FUNCTION_BLOCK "keller_pressure_transmitters"   // FB99, SCL
{ S7_Optimized_Access := 'TRUE' }
VERSION : 0.1
   VAR_INPUT
      mb_addr : USInt;
   END_VAR
   VAR_IN_OUT
      mb_query : "mb_query";
   END_VAR
   VAR
      sb : "mb_station_block_udt";
      data : Struct
         pressure_sensor_1 : Real;
         pressure_sensor_2 : Real;
         temperature : Real;
         temperature_sensor_1 : Real;
         temperature_sensor_2 : Real;
      END_STRUCT;
   END_VAR
BEGIN
   // Keller, Series 30 and Series 40 - Pressure transmitters
   // 
   // http://www.keller-druck.com/picts/pdf/engl/comm_protocol_e.pdf

   "mb_station_block_header"(sb := #sb,
                             mb_query := #mb_query);

   #mb_query(mb_addr := #mb_addr,
             mode := #mb_query.c.read.holding_reg,
             data_addr := 2,
             data_ptr := #data);

   "mb_station_block_footer"(sb := #sb,
                             mb_query := #mb_query);
END_FUNCTION_BLOCK

FUNCTION_BLOCK "Epever_solar_charge_controller"   // FB109, SCL
{ S7_Optimized_Access := 'TRUE' }
VERSION : 0.1
   VAR_INPUT
      mb_addr : UInt := 1;
      on : Bool;
   END_VAR
   VAR_OUTPUT
      PV_array_input_voltage : Real;
      PV_array_input_current : Real;
      PV_array_input_power : Real;
      battery_power : Real;
      load_voltage : Real;
      load_current : Real;
      load_power : Real;
      battery_temperature : Real;
      temperature_inside_equipment : Real;
      battery_soc : Real;   // The percentage of battery's remaining capacity
      remote_battery_temperature : Real;
      battery_real_rated_power : Real;
      _ : Bool;
      PV_voltage_today_Maximum : Real;
      PV_voltage_today_Minimum : Real;
      Battery_voltage_today_Maximum : Real;
      Battery_voltage_today_Minimum : Real;
      Consumed_energy_today : Real;
      Consumed_energy_this_month : Real;
      Consumed_energy_this_year : Real;
      Consumed_energy_total : Real;
      Generated_energy_today : Real;
      Generated_energy_this_month : Real;
      Generated_energy_this_year : Real;
      Generated_energy_total : Real;
      Battery_voltage : Real;
      Battery_current : Real;
      __ : Bool;
      charging_status : Struct
         No_charging : Bool;
         Float : Bool;
         Boost : Bool;
         Equalization : Bool;
      END_STRUCT;
   END_VAR
   VAR_IN_OUT
      mb_query : "mb_query";
   END_VAR
   VAR
      sb : "mb_station_block_udt";
      read3 : Struct
         load_short : Bool;   // [08]
         load_over_current : Bool;   // [09]
         Input_is_over_current : Bool;   // [10]
         Anti_reverse_MOSFET_is_short : Bool;   // [11]
         Charging_or_Anti_reverse_MOSFET_is_short : Bool;   // [12]
         Charging_MOSFET_is_short : Bool;   // [13]
         x14 : Bool;   // [14]
         x15 : Bool;   // [15]
         Running : Bool;   // [00] - Standby
         Normal : Bool;   // [01] - Fault
         charging_status_0 : Bool;   // [02]
         charging_status_1 : Bool;   // [03]
         PV_Input_is_short : Bool;   // [04]
         x05 : Bool;   // [05]
         x06 : Bool;   // [06]
         Load_MOSFET_is_short : Bool;   // [07]
      END_STRUCT;
      first_scan : Bool := true;
   END_VAR
   VAR_TEMP
      read1 : Struct
         PV_array_input_voltage : UInt;   // [3100]
         PV_array_input_current : UInt;   // [3101]
         PV_array_input_power : UDInt;   // [3102]
         z_1 : Array[1..3] of Word;
         battery_power : UDInt;   // [3106]
         z_2 : Array[1..4] of Word;
         load_voltage : UInt;   // [310C]
         load_current : UInt;   // [310D]
         load_power : UDInt;   // [310E]
         battery_temperature : UInt;   // [3110]
         temperature_inside_equipment : UInt;   // [3111]
         battery_soc : UInt;   // [311A] The percentage of battery's remaining capacity
         remote_battery_temperature : UInt;   // [311B]
         z_3 : UInt;
         battery_real_rated_power : UInt;   // [311D]
      END_STRUCT;
      read2 : Struct
         PV_voltage_today_Maximum : UInt;   // [3300]
         PV_voltage_today_Minimum : UInt;   // [3301]
         Battery_voltage_today_Maximum : UInt;   // [3302]
         Battery_voltage_today_Minimum : UInt;   // [3303]
         Consumed_energy_today : UDInt;   // [3304]
         Consumed_energy_this_month : UDInt;   // [3306]
         Consumed_energy_this_year : UDInt;   // [3308]
         Consumed_energy_total : UDInt;   // [330A]
         Generated_energy_today : UDInt;   // [330C]
         Generated_energy_this_month : UDInt;   // [330E]
         Generated_energy_this_year : UDInt;   // [3310]
         Generated_energy_total : UDInt;   // [3312]
         Battery_voltage : UInt;   // [331A]
         Battery_current : UDInt;   // [331B]
      END_STRUCT;
      tmp : Byte;
   END_VAR
BEGIN
   // Epever - solar charge controller 
   // v2.3 - 12 june 2015
   // 

   IF #first_scan THEN
       #sb.conf.read_only := true;
   END_IF;

   "mb_station_block_header"(sb := #sb, mb_query := #mb_query);
   #mb_query.mb_addr := #mb_addr; 

   #mb_query.mode := #mb_query.c.read.input_reg;
   #mb_query(data_addr := 16#3100, data_ptr := #read1);
   IF #mb_query.Done THEN
       #PV_array_input_voltage := UINT_TO_REAL(#read1.PV_array_input_voltage) / 100;
       #PV_array_input_current := UINT_TO_REAL(#read1.PV_array_input_current) / 100;
       #PV_array_input_power := UDINT_TO_REAL(ROR(IN := #read1.PV_array_input_power, N := 16)) / 100;
       #battery_power := UDINT_TO_REAL(ROR(IN := #read1.battery_power, N := 16)) / 100;
       #load_voltage := UINT_TO_REAL(#read1.load_voltage) / 100;
       #load_current := UINT_TO_REAL(#read1.load_current) / 100;
       #load_power := UDINT_TO_REAL(ROR(IN := #read1.load_power, N := 16)) / 100;
       #battery_temperature := UINT_TO_REAL(#read1.battery_temperature) / 100;
       #temperature_inside_equipment := UINT_TO_REAL(#read1.temperature_inside_equipment) / 100;
       #battery_soc := UINT_TO_REAL(#read1.battery_soc) / 100;
       #remote_battery_temperature := UINT_TO_REAL(#read1.remote_battery_temperature) / 100;
       #battery_real_rated_power := UINT_TO_REAL(#read1.battery_real_rated_power) / 100;
   END_IF;

   #mb_query(data_addr := 16#3300, data_ptr := #read2);
   IF #mb_query.Done THEN
       #PV_voltage_today_Maximum := UINT_TO_REAL(#read2.PV_voltage_today_Maximum) / 100;
       #PV_voltage_today_Minimum := UINT_TO_REAL(#read2.PV_voltage_today_Minimum) / 100;
       #Battery_voltage_today_Maximum := UINT_TO_REAL(#read2.Battery_voltage_today_Maximum) / 100;
       #Battery_voltage_today_Minimum := UINT_TO_REAL(#read2.Battery_voltage_today_Minimum) / 100;
       #Consumed_energy_today := UDINT_TO_REAL(ROR(IN := #read2.Consumed_energy_today, N := 16)) / 100;
       #Consumed_energy_this_month := UDINT_TO_REAL(ROR(IN := #read2.Consumed_energy_this_month, N := 16)) / 100;
       #Consumed_energy_this_year := UDINT_TO_REAL(ROR(IN := #read2.Consumed_energy_this_year, N := 16)) / 100;
       #Consumed_energy_total := UDINT_TO_REAL(ROR(IN := #read2.Consumed_energy_total, N := 16)) / 100;
       #Generated_energy_today := UDINT_TO_REAL(ROR(IN := #read2.Generated_energy_today, N := 16)) / 100;
       #Generated_energy_this_month := UDINT_TO_REAL(ROR(IN := #read2.Generated_energy_this_month, N := 16)) / 100;
       #Generated_energy_this_year := UDINT_TO_REAL(ROR(IN := #read2.Generated_energy_this_year, N := 16)) / 100;
       #Generated_energy_total := UDINT_TO_REAL(ROR(IN := #read2.Generated_energy_total, N := 16)) / 100;
       #Battery_voltage := UDINT_TO_REAL(#read2.Battery_voltage) / 100;
       #Battery_current := UDINT_TO_REAL(ROR(IN := #read2.Battery_current, N := 16)) / 100;
   END_IF;


   #mb_query(data_addr := 16#3201, data_ptr := #read3);
   #tmp.%X0 := #read3.charging_status_0;
   #tmp.%X1 := #read3.charging_status_1;
   #charging_status.No_charging := #tmp = 0;
   #charging_status.Float := #tmp = 1;
   #charging_status.Boost := #tmp = 2;
   #charging_status.Equalization := #tmp = 3;

   #mb_query.mode := #mb_query.c.write.single_discrete_output;
   #tmp.%X0 := #on;
   #mb_query(data_addr := 0, data_ptr := #tmp);

   "mb_station_block_footer"(sb := #sb, mb_query := #mb_query);


   (*
   - 16bit MODBUS addresses (per the modbus.org spec)
   - BPS: 115200 baud
   - Parity: None
   - Data bits: 8
   - Stop bits: 1
   - Flow control: None

   Pin definition RJ45 
   1   Power supply output +7.5
   2   Power supply output +7.5
   3   RS-485 - A
   4   RS-485 - A
   5   RS-485 - B
   6   RS-485 - B
   7   Ground
   8   Ground

   *)
END_FUNCTION_BLOCK

// folder: Library/Modbus/Station blocks/sb untested/Abb

FUNCTION_BLOCK "abb_aquaMaster_3"   // FB4, SCL
{ S7_Optimized_Access := 'TRUE' }
VERSION : 0.1
   VAR_INPUT
      mb_addr : USInt;
   END_VAR
   VAR_IN_OUT
      mb_query : "mb_query";
   END_VAR
   VAR
      sb : "mb_station_block_udt";
      flow : Real;
      pressure : Real;
      totaliser : Struct
         fwd : DInt;
         rev : DInt;
         net : DInt;
      END_STRUCT;
   END_VAR
BEGIN
   // - ABB - AquaMaster 3 - Electromagnetic flowmeter
   // - COI/FET2XX/MOD/TBLÃ¢â‚¬â€œEN
   // - https://library.e.abb.com/public/
   //   91eead459bb0d349c12577fc0033d2b5/COI_FET2XX_MOD_TBL-EN.pdf

   "mb_station_block_header"(sb := #sb, mb_query := #mb_query);
   #mb_query.mb_addr := #mb_addr; // Device address.

   // Two queries, reading input registers. 
   #mb_query.mode := #mb_query.c.read.input_reg;
   #mb_query(data_addr := 5017, data_ptr := #flow);
   #mb_query(data_addr := 5025, data_ptr := #pressure);

   // One query, reading one section of holding registers.
   #mb_query.mode := #mb_query.c.read.holding_reg;
   #mb_query(data_addr := 12003, data_ptr := #totaliser);

   // - Each query reading one section of holding registers.
   // - Data length is automatically calculated for holding 
   //   and input regisers.

   "mb_station_block_footer"(sb := #sb, mb_query := #mb_query);
END_FUNCTION_BLOCK

FUNCTION_BLOCK "Abb_266"   // FB12, SCL
{ S7_Optimized_Access := 'TRUE' }
VERSION : 0.1
   VAR_INPUT
      mb_addr : UInt;
   END_VAR
   VAR_IN_OUT
      mb_query : "mb_query";
   END_VAR
   VAR
      sb : "mb_station_block_udt";
      data : Struct
         "Differential Pressure" : Real;
         "Static Pressure" : Real;
         "Process Temperature" : Real;
         "Mass flow rate value" : Real;
         "Volume Flow rate value" : Real;
      END_STRUCT;
      settings : Struct
         Differential_Pressure_Units_Code : UInt := 12;
         Static_Pressure_Units_select_Code : UInt := 12;
         Temperature_Units_select_Code : UInt := 32;
      END_STRUCT;
   END_VAR
BEGIN
   // ABB - 266 MODBUS, multivariable transmitter.
   // Differential and Static Pressure, Temperature
   // 
   // https://library.e.abb.com/public/9b5a1233ec79400387d5b4887002fb00/2105216MNAA.pdf

   "mb_station_block_header"(sb := #sb, mb_query := #mb_query);
   #mb_query.mb_addr := #mb_addr;

   #mb_query(mode := #mb_query.c.read.holding_reg,
             data_addr := 401,
             data_ptr := #data);

   #mb_query(mode := #mb_query.c.write.holding_reg,
             data_addr := 481,
             data_ptr := #settings);

   "mb_station_block_footer"(sb := #sb, mb_query := #mb_query);

   (*
   Differential_Pressure_Units_Code
   1 = inches of water
   8 = Millibar (ROM default)
   11 = Pascal
   12 = Kilopascal 

   Static Pressure Units select Code
   6 = PSIA
   7 = Bar (ROM default)
   12 = Kilopascal
   117 = Megapascal 

   Temperature Units select Code
   32 = Degree Celsius (ROM default)
   33 = Degree Fahrenheit
   34 = Degree Rankine
   35 = Degree Kelvin

   *)
END_FUNCTION_BLOCK

FUNCTION_BLOCK "Abb_M2M_DMTME"   // FB15, SCL
{ S7_Optimized_Access := 'TRUE' }
VERSION : 0.1
   VAR_INPUT
      mb_addr : UInt;
   END_VAR
   VAR_IN_OUT
      mb_query : "mb_query";
   END_VAR
   VAR
      sb : "mb_station_block_udt";
      read1 : Struct
         "3-PHASE SYSTEM VOLTAGE" : UDInt;   // volt
         voltage_Lx_N : Array[1..3] of UDInt;   // volt
         voltage_L_L : Array[1..3] of UDInt;   // volt 1:L1-L2, 2:L2-L3, 3:L3-L1
         "3-PHASE SYSTEM CURRENT" : UDInt;
         current : Array[1..3] of UDInt;   // mA
         "3-PHASE SYS. POWER FACTOR" : DInt;   // x1000
         Power_factor : Array[1..3] of DInt;   // x1000
         "3-PHASE SYSTEM COS Ï•I" : DInt;   // x1000
         phase_cos : Array[1..3] of DInt;   // x1000
      END_STRUCT;
      read2 : Struct
         "3-PHASE S. APPARENT POWER" : UDInt;   // VA
         apparent_power : Array[1..3] of UDInt;   // VA
         "3-PHASE SYS. ACTIVE POWER" : DInt;   // Watt
         active_power : Array[1..3] of DInt;   // Watt
         "3-PHASE S. REACTIVE POWER" : UDInt;
         reactive_power : Array[1..3] of UDInt;
         "3-PHASE SYS. ACTIVE ENERGY" : UDInt;   // Wh * 100
         "3-PHASE S. REACTIVE ENERGY" : UDInt;   // VArh * 100
         frequency : UDInt;   // mHz
         "MAX LINE CURRENT" : Array[1..3] of UDInt;
      END_STRUCT;
   END_VAR
BEGIN
   // ABB - M2M/DMTME - 2CSG445011D0201 
   //
   // https://library.e.abb.com/public/3921770555944801ad6d9e002d23ca23/2CSG445011D0201.pdf

   "mb_station_block_header"(sb := #sb, mb_query := #mb_query);
   #mb_query.mb_addr := #mb_addr;

   #mb_query.mode := #mb_query.c.read.holding_reg;
   #mb_query(data_addr := 16#1000, data_ptr := #read1);
   #mb_query(data_addr := 16#1026, data_ptr := #read2);

   "mb_station_block_footer"(sb := #sb, mb_query := #mb_query);
END_FUNCTION_BLOCK

FUNCTION_BLOCK "Abb_ach_400_ac_drives"   // FB80, SCL
{ S7_Optimized_Access := 'TRUE' }
VERSION : 0.1
   VAR_INPUT
      mb_addr : UInt;
   END_VAR
   VAR_IN_OUT
      mb_query : "mb_query";
   END_VAR
   VAR
      sb : "mb_station_block_udt";
      read1 : Struct
         sw : Struct   // page 111, tabel 23
            x08_actual_eq_ref : Bool;   // (= is within tolerance limits)
            x09_drive_control_remote : Bool;
            x10_supervision_limit : Bool;   // The value of first supervised parameter equals to or is greater than supervision limit. Refer toGroup 32 Supervision.
            x11_ext2_selected : Bool;   // 0 = ext1 selected
            x12_run : Bool;   // Enable signal received
            x13 : Bool;
            x14 : Bool;
            x15 : Bool;
            x00_rdy_to_sw_on : Bool;
            x01_rdy_to_operate : Bool;
            x02_opr_enabled : Bool;
            x03_falut : Bool;
            x04_OFF2_inactive : Bool;
            x05_OFF3_inactive : Bool;
            x06_switch_on_innhibited : Bool;
            x07_alarm : Bool;   // See the Diagnostics section for a list of relevant alarms
         END_STRUCT;
      END_STRUCT;
      read2 : Struct
         speed : Int;   // rpm
         output_freq : Int;   // 0.1 Hz
         current : Int;   // 0.1 A
         torque : Int;   // 0.1 %
         power : Int;   // 0.1 kW
         dc_bus_voltage : Int;   // 0.1 V
         output_voltage : Int;   // 0.1 V
         ACH400_temp : Int;   // 0.1 Â°C | Displays the temperature of the ACH 400 heatsink in degrees Centigrade
         ext_ref_1 : Int;   // 0.1 Hz
         ext_ref_2 : Int;   // 0.1 %
         ctrl_location : Int;   // 0 - 2
         run_time : UInt;   // h
         kWh_cnt : UInt;   // kWh
         appl_blk_output : UInt;
         digital_input : Struct
            x08 : Bool;
            x09 : Bool;
            x10 : Bool;
            x11 : Bool;
            x12 : Bool;
            x13 : Bool;
            x14 : Bool;
            x15 : Bool;
            x00_in_1 : Bool;
            x01_in_2 : Bool;
            x02_in_3 : Bool;
            x03_in_4 : Bool;
            x04 : Bool;
            x05 : Bool;
            x06 : Bool;
            x07 : Bool;
         END_STRUCT;
         analog_in_1 : UInt;   // 0.1 %
         analog_in_2 : UInt;   // 0.1 %
      END_STRUCT;
      read3 : Struct
         fault_word_1 : Struct
            x08_Motor_overtemperature : Bool;
            x09_Panel_loss : Bool;
            x10_Parameters_inconsistent : Bool;
            x11_DC_bus_ripple_too_large : Bool;
            x12_Motor_stall : Bool;
            x13_Serial_communication_loss : Bool;
            x14_External_fault : Bool;
            x15_Output_ground_fault : Bool;
            x00_Overcurrent : Bool;
            x01_DC_overvoltage : Bool;
            x02_ACH_400_overtemperature : Bool;
            x03_Fault_current : Bool;
            x04_Output_overload : Bool;
            x05_DC_undervoltage : Bool;
            x06_Analog_input_1_fault : Bool;
            x07_Analog_input_2_fault : Bool;
         END_STRUCT;
         fault_word_2 : Struct
            x08_hw_err : Bool;
            x09_hw_err : Bool;
            x10_hw_err : Bool;
            x11_hw_err : Bool;
            x12_hw_err : Bool;
            x13_hw_err : Bool;
            x14_hw_err : Bool;
            x15_hw_err : Bool;
            x00_Underload : Bool;
            x01 : Bool;
            x02_DDCS_link : Bool;
            x03 : Bool;
            x04 : Bool;
            x05 : Bool;
            x06 : Bool;
            x07 : Bool;
         END_STRUCT;
      END_STRUCT;
      _ : Bool;
      write1 : Struct
         cw : Struct   // page 109, tabel 21
            x08 : Bool;
            x09 : Bool;
            x10 : Bool;
            x11_sel_ext_2 : Bool;   // Select external control location 1
            x12 : Bool;
            x13 : Bool;
            x14 : Bool;
            x15 : Bool;
            x00_start : Bool := TRUE;
            x01_no_cost_stop : Bool := TRUE;   // Emergency OFF, coast to stop.Enter OFF2 ACTIVE; proceed to SWITCH-ON INHIBITED
            x02_no_ramp_stop : Bool := TRUE;   // Emergency stop. Drive ramps to stop according to parameter 2205 DECELER TIME 2. Enter
            x03_operation_enable : Bool := TRUE;
            x04 : Bool;
            x05_no_ramp_generator : Bool := TRUE;
            x06_no_force_ramp_generator_input2zero : Bool;   // Force Ramp Function Generator input to zero
            x07_fault_reset : Bool;   // (enter SWITCH-ON INHIBITED)
         END_STRUCT;
         ref_1 : Int;
         ref_2 : Int;
      END_STRUCT;
      write2 : Struct
         keypad_ref_sel : UInt;
         ext1_ext2_sel : UInt;
         ext1_sel : UInt;
         ext1_sel_min : UInt;   // 0 - 250 Hz
         ext1_sel_max : UInt := 50;   // 0 - 250 Hz
      END_STRUCT;
      write3 : Struct   // Communication fault function
         comm_fault_func : UInt := 1;   // 1=FAULT(cost), 2=CONST SP 7, 3=LAST SPEED
      END_STRUCT;
   END_VAR
BEGIN
   // Abb - ACH 400 - AC Drives 
   // 
   // Web: https://www.ccontrols.com/support/dp/ACH402_US_04_Web.pdf

   "mb_station_block_header"(sb := #sb, mb_query := #mb_query);
   #mb_query.mb_addr := #mb_addr;

   #mb_query.mode := #mb_query.c.read.holding_reg;
   #mb_query(data_addr := 3, data_ptr := #read1);   // 40004
   #mb_query(data_addr := 102, data_ptr := #read2); // 103
   #mb_query(data_addr := 304, data_ptr := #read3); // 305 - 1 

   #mb_query.mode := #mb_query.c.write.holding_reg;
   #mb_query(data_addr := 0, data_ptr := #write1); // 40001
   // #mb_query(data_addr := 1100, data_ptr := #write2); // 1101 - 1
   #mb_query(data_addr := 5003, data_ptr := #write3); // 5004 - 1

   "mb_station_block_footer"(sb := #sb, mb_query := #mb_query);
END_FUNCTION_BLOCK

// folder: Library/Modbus/Station blocks/sb untested/Floridan

FUNCTION_BLOCK "Floridan_Uniflo_1200"   // FB83, SCL
{ S7_Optimized_Access := 'TRUE' }
VERSION : 0.1
   VAR_INPUT
      mb_addr : USInt;
      delay : Time := T#10S;
   END_VAR
   VAR_OUTPUT
      energi : LReal;   // [MJ]
      vol_measured : LReal;   // [m3]
      vol_conv : LReal;   // [Nm3]
      pressure : LReal;   // [bar A]
      temperature : LReal;
   END_VAR
   VAR_IN_OUT
      mb_query : "mb_query";
   END_VAR
   VAR
      sb : "mb_station_block_udt";
      battery_remaining : UInt;
      mb_delay : "mb_delay";
      serial_number : String[6];
   END_VAR
   VAR_TEMP
      dommy : Bool;
      c : Int;
      "dword" : DWord;
   END_VAR
BEGIN
   // Flonidan - Uniflo 1200 GVEC
   // Product number: 061864X-YYY
   //
   // - https://www.gavilar.nl/files/communicationboard230210_1521630740_b6a3b533.pdf
   // - M/06180XX/24

   "mb_station_block_header"(sb := #sb, mb_query := #mb_query);
   #mb_query.mb_addr := #mb_addr; // Device address.

   // Reduce power consumption, by halting execution. Nice if the device is running 
   // on battery. mb_delay is located inside the mb_extended_features.scl file.
   #mb_delay(delay := #delay, mb_query := #mb_query);

   #mb_query.mb_addr.%X5 := 0; // - Last bits of mb_addr is used for expanding 
   #mb_query.mb_addr.%X6 := 0; //   register addr, this means that only addr 1
   #mb_query.mb_addr.%X7 := 0; //   to 31 on the bus may be used.

   #mb_query.mode := #mb_query.c.read.holding_reg;

   #mb_query(data_addr := 123, data_ptr := #battery_remaining);
   #mb_query(data_addr := 2833, data_ptr := #serial_number); // Serial number 

   #mb_query.conf.buffer_handler := false;

   #mb_query(data_addr := 56, data_len := 44, data_ptr := #dommy);
   IF #mb_query.Done THEN
       #vol_conv := "intreal"(mb_query := #mb_query, addr := 16#70 / 2);
       #"dword".%B3 := #mb_query.z.buffer[16]; // 16#80/2=64, (64-56)*2=16
       #"dword".%B2 := #mb_query.z.buffer[17];
       #"dword".%B1 := #mb_query.z.buffer[18];
       #"dword".%B0 := #mb_query.z.buffer[19];
       #pressure := DWORD_TO_REAL(#"dword");
       #"dword".%B3 := #mb_query.z.buffer[20]; // 16#84/2=66, (66-56)*2=20
       #"dword".%B2 := #mb_query.z.buffer[21];
       #"dword".%B1 := #mb_query.z.buffer[22];
       #"dword".%B0 := #mb_query.z.buffer[23];
       #temperature := DWORD_TO_REAL(#"dword");
       #energi := "intreal"(mb_query := #mb_query, addr := 16#90 / 2);
       #vol_measured := "intreal"(mb_query := #mb_query, addr := 16#98 / 2);
   END_IF;

   #mb_query.data_len := #mb_query.c.auto_len;
   #mb_query.conf.buffer_handler := true;
   "mb_station_block_footer"(sb := #sb, mb_query := #mb_query);
END_FUNCTION_BLOCK

FUNCTION "intreal" : LReal   // FC16, SCL
{ S7_Optimized_Access := 'TRUE' }
VERSION : 0.1
   VAR_INPUT
      mb_query : "mb_query";
      addr : UInt;
   END_VAR
   VAR_TEMP
      dw : UDInt;
      r : DWord;
      bo : UDInt;
   END_VAR
BEGIN
   // Uniflo 1200 has a special datatype named
   // int-real, this block decode that data type.

   // buffer offset
   #bo := (#addr - #mb_query.data_addr) * 2;

   // The integer part of the value, little endian.
   #dw.%B3 := #mb_query.z.buffer[#bo + 0];
   #dw.%B2 := #mb_query.z.buffer[#bo + 1];
   #dw.%B1 := #mb_query.z.buffer[#bo + 2];
   #dw.%B0 := #mb_query.z.buffer[#bo + 3];
   #intreal := UDINT_TO_LREAL(#dw);

   // The decimal part of the value, little endian.
   // Stored as a real (IEEE754).
   #r.%B3 := #mb_query.z.buffer[#bo + 4];
   #r.%B2 := #mb_query.z.buffer[#bo + 5];
   #r.%B1 := #mb_query.z.buffer[#bo + 6];
   #r.%B0 := #mb_query.z.buffer[#bo + 7];
   #intreal += DWORD_TO_REAL(#r);
END_FUNCTION

// folder: Library/Modbus/Station blocks/sb untested/Grundfoss

FUNCTION_BLOCK "Grunnfoss_pump"   // FB14, SCL
{ S7_Optimized_Access := 'TRUE' }
VERSION : 0.1
   VAR_INPUT
      mb_addr : USInt;
      setpoint : Real;   // [%]
   END_VAR
   VAR_OUTPUT
      ProcessFeedback : Real;
      _ : Bool;
      Head : Real;   // bar
      VolumeFlow : Real;   // m3/h
      RelativePerformance : Real;   // %
      Speed : Real;   // rpm
      Frequency : Real;   // Hz
      ActualSetpoint : Real;   // %
      MotorCurrent : Real;   // A
      DCLinkVoltage : Real;   // V
      MotorVoltage : Real;   // V
      Power : Real;   // W
      RemoteFlow : Real;   // m3/h
      InletPressure : Real;   // bar
      RemotePressure : Real;   // bar
      Level : Real;   // m
      PowerElectronicTemp : Real;   // degree C
      MotorTemp : Real;   // degree C
      RemoteTemp : Real;   // degree C
      ElectronicTemp : Real;   // degree C
      PumpLiquidTemp : Real;   // degree C
      BearingTempDE : Real;   // degree C
      BearingTempNDE : Real;   // degree C
      AuxSensorInput : Real;   // %
      SpecificEnergyConsumption : Real;   // Wh/m3
      OperationTime : Real;   // hour
      TotalPoweredTime : Real;   // hour
      Torque : Real;   // Nm
      Energy : Real;   // kWh
      NumberOfStarts : Real;
   END_VAR
   VAR_IN_OUT
      mb_query : "mb_query";
   END_VAR
   VAR
      sb : "mb_station_block_udt";
      read1 : Struct
         status : Struct   // (201)
            x08_AccessModeRemote : Bool;
            x09_On : Bool;
            x10_Fault : Bool;
            x11_Warning : Bool;
            x12_ForcedToLocal : Bool;
            x13_AtMaxSpeed : Bool;
            x14 : Bool;
            x15_AtMinSpeed : Bool;
            x00_LowFlowStop : Bool;
            x01_CopyToLocal : Bool;
            x02_MaxFlowLimitEnabled : Bool;
            x03_ResetAlarmAck : Bool;
            x04_SetpointInfluence : Bool;
            x05_AtMaxPower : Bool;
            x06_Rotation : Bool;
            x07_Direction : Bool;
         END_STRUCT;
         ProcessFeedback : UInt;   // (202) x 0.01
         ControlMode : UInt;   // (203)
         OperationMode : UInt;   // (204)
         AlarmCode : UInt;   // (205)
         WarningCode : UInt;   // (206)
         MonthsToBearingService : Byte;   // (207)
         BearingServiceType : Byte;
         DriveState : UInt;   // (208)
         FeedbackSensorUnit : UInt;   // (209)
         FeedbackSensorMin : UInt;   // (210)
         FeedbackSensorMax : UInt;   // (211)
         NominalFrequency : UInt;   // (212)
         MinFrequency : UInt;   // (213) Minimum frequency in % of nominal frequency
         MaxFrequency : UInt;   // (214) Maximum frequency in % of nominal frequency
         SetpointRangeMin : UInt;   // (215)
         SetpointRangeMax : UInt;   // (216)
         _ : Array[1..4] of UInt;
         FlowEstimationState : UInt;   // (221) 0: within range, 1:below, 2:above
      END_STRUCT;
      read2 : Struct
         Head : UInt;   // (301) 0.001 bar
         VolumeFlow : UInt;   // (302) 0.1 m3/h
         RelativePerformance : UInt;   // (303) 0.01 %
         Speed : UInt;   // (304) rpm
         Frequency : UInt;   // (305) 0.1 Hz
         DigitalInput : Word;   // (306)
         DigitalOutput : Word;   // (307)
         ActualSetpoint : UInt;   // (308) 0.01 %
         MotorCurrent : UInt;   // (309) 0.1 A
         DCLinkVoltage : UInt;   // (310) 0.1 V
         MotorVoltage : UInt;   // (311) 0.1 V
         Power : UDInt;   // (312) W
         RemoteFlow : UInt;   // (314) 0.1 m3/h
         InletPressure : UInt;   // (315) 0.001 bar
         RemotePressure : UInt;   // (316) 0.001 bar
         Level : UInt;   // (317) 0.01 m
         PowerElectronicTemp : UInt;   // (318) 0.01 K
         MotorTemp : UInt;   // (319) 0.01 K
         RemoteTemp : UInt;   // (320) 0.01 K
         ElectronicTemp : UInt;   // (321) 0.01 K
         PumpLiquidTemp : UInt;   // (322) 0.01 K
         BearingTempDE : UInt;   // (323) 0.01 K
         BearingTempNDE : UInt;   // (324) 0.01 K
         AuxSensorInput : UInt;   // (325) 0.01 %
         SpecificEnergyConsumption : UInt;   // (326) Wh/m3
         OperationTime : UDInt;   // (327) hour
         TotalPoweredTime : UDInt;   // (329) hour
         Torque : UInt;   // (331) 0.1 Nm
         Energy : UDInt;   // (332) kWh
         NumberOfStarts : UDInt;   // (334)
      END_STRUCT;
      write : Struct
         cmd : Struct   // (101)
            x08 : Bool;
            x09 : Bool;
            x10 : Bool;
            x11 : Bool;
            x12 : Bool;
            x13 : Bool;
            x14 : Bool;
            x15 : Bool;
            x00_Remote : Bool := true;   // 0=Local
            x01_On : Bool;   // 0=Off
            x02_ResetAlarm : Bool;   // rising edge only
            x03_CopyToLocal : Bool;
            x04_EnableMaxFlowLimit : Bool;
            x05 : Bool;
            x06 : Bool;
            x07 : Bool;
         END_STRUCT;
         ControlMode : UInt;   // (102)
         OperationMode : UInt;   // (103)
         Setpoint : UInt;   // (104)
         Relay : Struct   // (105)
            x08 : Bool;
            x09 : Bool;
            x10 : Bool;
            x11 : Bool;
            x12 : Bool;
            x13 : Bool;
            x14 : Bool;
            x15 : Bool;
            x00_Realy1_inverted : Bool;   // 0: Closed, 1:Open
            x01_Realy2_inverted : Bool;   // 0: Closed, 1:Open
            x02_Realy3_inverted : Bool;   // 0: Closed, 1:Open
            x03_Realy4_inverted : Bool;   // 0: Closed, 1:Open
            x04 : Bool;
            x05 : Bool;
            x06 : Bool;
            x07 : Bool;
            x : Struct
               x08 : Bool;
               x09 : Bool;
               x10 : Bool;
               x11 : Bool;
               x12 : Bool;
               x13 : Bool;
               x14 : Bool;
               x15 : Bool;
               x00 : Bool;
               x01 : Bool;
               x02 : Bool;
               x03 : Bool;
               x04 : Bool;
               x05 : Bool;
               x06 : Bool;
               x07 : Bool;
            END_STRUCT;
            x_1 : Struct
               x08 : Bool;
               x09 : Bool;
               x10 : Bool;
               x11 : Bool;
               x12 : Bool;
               x13 : Bool;
               x14 : Bool;
               x15 : Bool;
               x00 : Bool;
               x01 : Bool;
               x02 : Bool;
               x03 : Bool;
               x04 : Bool;
               x05 : Bool;
               x06 : Bool;
               x07 : Bool;
               x : Struct
                  x08 : Bool;
                  x09 : Bool;
                  x10 : Bool;
                  x11 : Bool;
                  x12 : Bool;
                  x13 : Bool;
                  x14 : Bool;
                  x15 : Bool;
                  x00 : Bool;
                  x01 : Bool;
                  x02 : Bool;
                  x03 : Bool;
                  x04 : Bool;
                  x05 : Bool;
                  x06 : Bool;
                  x07 : Bool;
               END_STRUCT;
            END_STRUCT;
         END_STRUCT;
         SetMaxFlowLimit : UInt;   // (106) 0.01 m3/h
      END_STRUCT;
   END_VAR
BEGIN
   // Grundfoss - Pumps
   // CIM 200 Modbus RTU
   // CIM 500 Modbus TCP

   "mb_station_block_header"(sb := #sb, mb_query := #mb_query);
   #mb_query.mb_addr := #mb_addr;

   #mb_query.mode := #mb_query.c.read.holding_reg;

   #mb_query(data_addr := 201, data_ptr := #read1);
   IF #mb_query.Done THEN
       #ProcessFeedback := UINT_TO_REAL(#read1.ProcessFeedback) / 100;
   END_IF;

   #mb_query(data_addr := 301, data_ptr := #read2);
   IF #mb_query.Done THEN
       #Head := UINT_TO_REAL(#read2.Head) * 0.001;
       #VolumeFlow := UINT_TO_REAL(#read2.VolumeFlow) * 0.1;
       #RelativePerformance := UINT_TO_REAL(#read2.RelativePerformance) * 0.01;
       #Speed := UINT_TO_REAL(#read2.Speed);
       #Frequency := UINT_TO_REAL(#read2.Frequency) * 0.1;
       #ActualSetpoint := UINT_TO_REAL(#read2.ActualSetpoint) * 0.01;
       #MotorCurrent := UINT_TO_REAL(#read2.MotorCurrent) * 0.1;
       #DCLinkVoltage := UINT_TO_REAL(#read2.DCLinkVoltage) * 0.1;
       #MotorVoltage := UINT_TO_REAL(#read2.MotorVoltage) * 0.1;
       #Power := UDINT_TO_REAL(#read2.Power);
       #RemoteFlow := UINT_TO_REAL(#read2.RemoteFlow) * 0.1;
       #InletPressure := UINT_TO_REAL(#read2.InletPressure) * 0.001;
       #RemotePressure := UINT_TO_REAL(#read2.RemotePressure) * 0.001;
       #Level := UINT_TO_REAL(#read2.Level) * 0.01;
       #PowerElectronicTemp := UINT_TO_REAL(#read2.PowerElectronicTemp) * 0.01 - 273.15;
       #MotorTemp := UINT_TO_REAL(#read2.MotorTemp) * 0.01 - 273.15;
       #RemoteTemp := UINT_TO_REAL(#read2.RemoteTemp) * 0.01 - 273.15;
       #ElectronicTemp := UINT_TO_REAL(#read2.ElectronicTemp) * 0.01 - 273.15;
       #PumpLiquidTemp := UINT_TO_REAL(#read2.PumpLiquidTemp) * 0.01 - 273.15;
       #BearingTempDE := UINT_TO_REAL(#read2.BearingTempDE) * 0.01 - 273.15;
       #BearingTempNDE := UINT_TO_REAL(#read2.BearingTempNDE) * 0.01 - 273.15;
       #AuxSensorInput := UINT_TO_REAL(#read2.AuxSensorInput) * 0.01;
       #SpecificEnergyConsumption := UINT_TO_REAL(#read2.SpecificEnergyConsumption);
       #OperationTime := UDINT_TO_REAL(#read2.OperationTime);
       #TotalPoweredTime := UDINT_TO_REAL(#read2.TotalPoweredTime);
       #Torque := UINT_TO_REAL(#read2.Torque) * 0.1;
       #Energy := UDINT_TO_REAL(#read2.Energy);
       #NumberOfStarts := UDINT_TO_REAL(#read2.NumberOfStarts);
   END_IF;


   // Write preparations
   #write.cmd.x01_On := #setpoint <> 0;
   #write.Setpoint := REAL_TO_UINT(#setpoint * 100);

   #mb_query.mode := #mb_query.c.write.holding_reg;
   #mb_query(data_addr := 101, data_ptr := #write);

   "mb_station_block_footer"(sb := #sb, mb_query := #mb_query);

   (*

   #write.ControlMode:
   Some modes are not supported by all E-pumps.
   0: Constant speed
   1: Constant frequency
   3: Constant head
   4: Constant pressure
   5: Constant differential pressure
   6: Proportional pressure
   7: Constant flow
   8: Constant temperature
   10: Constant level
   128: AUTOADAPT
   129: FLOWADAPT (set FLOWLIMIT in register 00106)
   130: Closed-loop sensor.

   #write.OperationMode:
   0: Auto-control (setpoint control according to selected control mode)
   4: OpenLoopMin (running at minimum speed)
   6: OpenLoopMax (running at maximum speed)

   #read.DriveState:
   0: Stopped
   1: Accelerating
   2: Decelerating
   3: Steady state/closed loop
   4: -
   5: Accelerating halt
   6: Decelerating halt
   7: Start on the run (flying cut-in)
   Only MGE motors and CUE drives.

   #read.FeedbackSensorUnit:
   0: bar
   1: mbar
   2: m
   3: kPa
   4: psi
   5: ft
   6: m3/h
   7: m3/s
   8: l/s
   9: gpm
   10: °C
   11: °F
   12: %
   13: K
   14: W

   *)
END_FUNCTION_BLOCK

// folder: Library/Modbus/Station blocks/sb untested/Honeywell

FUNCTION_BLOCK "Honeywell_UDA2182"   // FB28, SCL
{ S7_Optimized_Access := 'TRUE' }
VERSION : 0.1
   VAR_INPUT
      mb_addr : UInt;
   END_VAR
   VAR_IN_OUT
      mb_query : "mb_query";
   END_VAR
   VAR
      sb : "mb_station_block_udt";
      data : Struct
         pv1 : Array[1..2] of Real;
         temperature : Array[1..2] of Real;
         alarm : Array[1..4] of DWord;
      END_STRUCT;
   END_VAR
BEGIN
   // Honeywell - UDA2182
   // 
   // Web: https://www.honeywellprocess.com/library/support/Public/Documents/70-82-25-126.pdf

   "mb_station_block_header"(sb := #sb, mb_query := #mb_query);
   #mb_query.mb_addr := #mb_addr;

   #mb_query.mode := #mb_query.c.mode.read;
   #mb_query(data_addr := 30001, data_ptr := #data);

   "mb_station_block_footer"(sb := #sb, mb_query := #mb_query);
END_FUNCTION_BLOCK

FUNCTION_BLOCK "Honeywell_variable_frequency_drives"   // FB29, SCL
{ S7_Optimized_Access := 'TRUE' }
VERSION : 0.1
   VAR_INPUT
      mb_addr : UInt := 255;
   END_VAR
   VAR_IN_OUT
      mb_query : "mb_query";
   END_VAR
   VAR
      sb : "mb_station_block_udt";
      read : Struct
         stw : Struct
            x24 : Bool;
            x25 : Bool;
            x26 : Bool;
            x27 : Bool;
            x28 : Bool;
            x29_control_place : Bool := FALSE;
            x30_control_place : Bool := FALSE;
            x31_control_place : Bool := TRUE;
            x16 : Bool;
            x17 : Bool;
            x18 : Bool;
            x19 : Bool;
            x20 : Bool;
            x21 : Bool;
            x22 : Bool;
            x23 : Bool;
            x08 : Bool;
            x09 : Bool;
            x10 : Bool;
            x11 : Bool;
            x12 : Bool;
            x13 : Bool;
            x14 : Bool;
            x15 : Bool;
            x00_Ready : Bool;
            x01_Running : Bool;
            x02_Counterclockwise : Bool;
            x03_Faulted : Bool;
            x04_Alarm : Bool;
            x05_AtReference : Bool;
            x06_ZeroSpeed : Bool;
            x07_FluxReady : Bool;
         END_STRUCT;
         d1_Output_Frequency : DInt;   // 0,01 Hz
         d2_Motor_Speed : DInt;   // 1 rpm
         d3_Motor_Current : DInt;   // 0,1 A
         d4_Motor_Torque : DInt;   // 0,1 %
         d5_Motor_Power : DInt;   // 0,1 %
         d6_Motor_Voltage : DInt;   // 0,1 V
         d7_DC_link_voltage : DInt;   // 1 V
         d8_Active_Fault_Code : DInt;
      END_STRUCT;
      write : Struct
         ctw : Struct
            x08 : Bool;
            x09 : Bool;
            x10 : Bool;
            x11 : Bool;
            x12 : Bool;
            x13 : Bool;
            x14 : Bool;
            x15 : Bool;
            x00 : Bool;
            x01_start : Bool := TRUE;
            x02_Reverse : Bool;
            x03_Reset_faults : Bool;
            x04 : Bool;
            x05 : Bool;
            x06 : Bool;
            x07 : Bool;
         END_STRUCT;
         __ : Word;
         speed_ref : UInt;   // 0â€¦10000 %
      END_STRUCT;
   END_VAR
BEGIN
   // Honeywell - Variable frequency drives
   // 
   // Web: https://customer.honeywell.com/resources/techlit/
   //      TechLitDocuments/62-0000s/62-0351.pdf

   "mb_station_block_header"(sb := #sb, mb_query := #mb_query);
   #mb_query.mb_addr := #mb_addr;

   #mb_query(mode := #mb_query.c.read.holding_reg,
             data_addr := 2151,
             data_ptr := #read);

   #mb_query(mode := #mb_query.c.write.holding_reg,
             data_addr := 2001,
             data_ptr := #write);

   "mb_station_block_footer"(sb := #sb, mb_query := #mb_query);
END_FUNCTION_BLOCK

// folder: Library/Modbus/Station blocks/sb untested/Krohne

FUNCTION_BLOCK "Krohne_Optisonic"   // FB34, SCL
{ S7_Optimized_Access := 'TRUE' }
VERSION : 0.1
   VAR_INPUT
      mb_addr : UInt;
   END_VAR
   VAR_IN_OUT
      mb_query : "mb_query";
   END_VAR
   VAR
      sb : "mb_station_block_udt";
      data : Struct
         "Temperature process value" : Real;
         "Dynamic Viscosity at Process conditions" : Real;
         "Density Process" : Real;
         "Flow Process" : Real;
         "Velocity Process" : Real;
         "Speed of Sound" : Real;
      END_STRUCT;
   END_VAR
BEGIN
   // Krohne - Optisonic V6
   // 

   "mb_station_block_header"(sb := #sb,
                             mb_query := #mb_query);
   #mb_query.mb_addr := #mb_addr;

   #mb_query.mode := #mb_query.c.read.holding_reg;
   #mb_query(data_addr := 7050,
             data_ptr := #data);

   "mb_station_block_footer"(sb := #sb,
                             mb_query := #mb_query);
END_FUNCTION_BLOCK

FUNCTION_BLOCK "Krohne_MFC_300"   // FB100, SCL
TITLE = Krohne MFC 300
{ S7_Optimized_Access := 'TRUE' }
AUTHOR : OlaBjornli
FAMILY : modbus
VERSION : 0.1
// Coriolise flow meter
   VAR_INPUT
      mb_addr : UInt;
   END_VAR
   VAR_OUTPUT
      Temperature : Real;   // [degree C]
   END_VAR
   VAR_IN_OUT
      mb_query : "mb_query";
   END_VAR
   VAR
      sb : "mb_station_block_udt";
      read1 : Struct
         "Flow Velocity" : Real;   // [m/s]
         "Volume Flow" : Real;   // [m3/s]
         "Mass Flow" : Real;   // [kg/s]
         Temperature : Real := 273.15;   // [K]
         Density : Real;   // [kg/m3]
         Concentration_1 : Real;
         Concentration_2_or_Diagnosis_3 : Real;
         Concentration_Flow_1 : Real;
         Concentration_Flow_2 : Real;
         Diagnosis_1 : Real;
         Diagnosis_2 : Real;
         Display_Channel_1 : Real;
         Display_Channel_2 : Real;
         Operating_time : Real;   // [s]
      END_STRUCT;
      write1_settings : Struct
         Counter_1_Function : UInt;
         Counter_1_Measurement : UInt;
         Counter_2_Function : UInt;
         Counter_2_Measurement : UInt;
         Counter_3_Function : UInt;
         Counter_3_Measurement : UInt;
      END_STRUCT;
      exec_write : Bool;
   END_VAR
BEGIN
   // Krohne - MFC 300 
   // Flowmeter
   // 
   // Web: http://cdn.krohne.com/dlc/AD_MFC300_Modbus_en_091124_4000744801_R01.pdf
   //
   // #settings :
   //    Counter Function:
   //       1 = Sum Counter
   //       2 = + Counter
   //       3 = - Counter
   //       0 = Off
   //    Counter Measurement:
   //       21 = Volume Flow [m3]
   //       22 = Mass Flow [kg]
   //       27 = Concentration Flow 1
   //       28 = Concentration Flow 2

   "mb_station_block_header"(sb := #sb, mb_query := #mb_query);
   #mb_query.mb_addr := #mb_addr;

   #mb_query(mode := #mb_query.c.mode.read,
             data_addr := 30001, // 30000 + 1 (error in datasheet)
             data_ptr := #read1);
   #Temperature := #read1.Temperature - 273.15;

   // The write query isn't executing continuously in case that will damage eeprom
   IF #exec_write THEN
       #mb_query(mode := #mb_query.c.mode.write,
                 data_addr := 40001, // 40000 + 1,
                 data_ptr := #write1_settings);
       #exec_write := NOT #mb_query.Done;
   END_IF;

   "mb_station_block_footer"(sb := #sb, mb_query := #mb_query);
END_FUNCTION_BLOCK

// folder: Library/Modbus/Station blocks/sb untested/Mettler

FUNCTION_BLOCK "mettler_toledo_IND560_loadTargetValue"   // FB87, SCL
{ S7_Optimized_Access := 'TRUE' }
VERSION : 0.1
   VAR_INPUT
      iValue : Real;
   END_VAR
   VAR_OUTPUT
      qDone : Bool;
   END_VAR
   VAR_IN_OUT
      "M" : "mettlerToledoInd560Udt";
      sb : "mb_station_block_udt";
   END_VAR
   VAR
      state : Int;
      old_value : Real;
      slot : USInt;
   END_VAR
   VAR CONSTANT
      NONE_AVAILABLE : USInt := 0;
   END_VAR
BEGIN
   // Load target value, for scale 1. Page 143, table B-6

   CASE #state OF

       0:  // Waiting for start.
           #qDone := false;
           #state +=
           BOOL_TO_INT(#old_value <> #iValue);

       1:  // Wait for available msg. slot
           #slot := "reqMsgSlot"(#"M".occupiedMsgSlots);
           #state += BOOL_TO_INT(#slot <> #NONE_AVAILABLE);

       2:  // #1 PLC loads floating point value first
           #"M".writeMsgSlot[#slot].cmd := 0;
           #"M".writeMsgSlot[#slot].data := #iValue;
           #state += 1;
       3:
           #state += BOOL_TO_INT(#"M".queryDone.write);

       4:  // #2 PLC sends command to set target 1 cutoff value 
           #"M".writeMsgSlot[#slot].cmd := 110;
           #state += 1;
       5:
           #state += BOOL_TO_INT(#"M".queryDone.write);

       6:  // #3 IND560 terminal sees new command, loads the value into the target
           //    and ends a return message to indicate the new target value.
           #state +=
           BOOL_TO_INT(#"M".queryDone.read
                       AND #"M".run.cmdAck[#slot] = 1
                       AND #"M".run.PF[#slot] = 13
                       AND #"M".readMsgSlot[#slot].data = #"M".writeMsgSlot[#slot].data);

       7:  // #4  PLC instructs IND560 terminal to start â€œusingâ€ new target value
           #"M".writeMsgSlot[#slot].cmd := 114;
           #state += 1;
       8:
           #state += BOOL_TO_INT(#"M".queryDone.write);

       9:  // #5 IND560 terminal sees new command
           #"M".writeMsgSlot[#slot].cmd := 0;

           #state +=
           BOOL_TO_INT(#"M".queryDone.read
                       AND #"M".run.cmdAck[#slot] = 2
                       AND #"M".run.PF[#slot] = 30
                       AND #"M".readMsgSlot[#slot].data = 0);

       ELSE: // Back to start.
           #"M".occupiedMsgSlots[#slot] := false; // Release msg. slot.
           #state := 0;
           #qDone := true;
           // The start signal should need to be set back false before next
           // exec. else the sequence will start over.
   END_CASE;
   #old_value := #iValue;

   // 
   IF #sb.out.communication_error THEN
       #state := 0;
       IF #slot <> #NONE_AVAILABLE THEN
           #"M".writeMsgSlot[#slot].cmd := 0;
           "releaseMsgSlot"(slot := #slot,
                            mem := #"M".occupiedMsgSlots);
       END_IF;
   END_IF;
END_FUNCTION_BLOCK

FUNCTION_BLOCK "mettler_toledo_IND560"   // FB88, SCL
{ S7_Optimized_Access := 'TRUE' }
VERSION : 0.1
   VAR_IN_OUT
      mb_query : "mb_query";
   END_VAR
   VAR
      mb_addr : UInt := 255;
      sb : "mb_station_block_udt";
      "M" : "mettlerToledoInd560Udt";   // Shared data
      loadTargetValue : "mettler_toledo_IND560_loadTargetValue";
      s : USInt;
   END_VAR
   VAR_TEMP
      c : Int;
   END_VAR
BEGIN
   // Mettler Toledo IND560 - Weighing Terminal

   // WARNING: This SB is just a draft and the block probably include errors !!

   // Necessary settings: ()
   // PLC -> Eth/IP - Modbus TCP -> IP-address
   // PLC -> Eth/IP - Modbus TCP -> Subnet-mask
   // PLC -> Data Format -> Byte order : standard
   // PLC -> Data Format -> Format     : Floating Point 

   // - Modbus tcp:
   //   https://bradysystems.com/wp-content/uploads/2012/10/IND560-PLC-Interface-Manual.pdf
   // - Product overview:
   //   http://www.atsackfillers.mobi/assets/ind560_ug_en_71209396_r04.pdf

   REGION Modbus
       "mb_station_block_header"(sb := #sb,
                                 mb_query := #mb_query);
       #mb_query.mb_addr := #mb_addr;

       #mb_query(mode := #mb_query.c.mode.read,
                 data_addr := 400001,
                 data_ptr := #"M".readMsgSlot,
                 Done => #"M".queryDone.read);

       #mb_query(mode := #mb_query.c.mode.write,
                 data_addr := 401026,
                 data_ptr := #"M".writeMsgSlot,
                 Done => #"M".queryDone.write);

       "mb_station_block_footer"(sb := #sb,
                                 mb_query := #mb_query);
   END_REGION

   REGION Read data-fix     
       // Extract bits in word in to a numbers.
       FOR #c := 1 TO 4 DO
           #"M".run.PF[#c].%X0 := #"M".readMsgSlot[#c].cmdRespons.FP_1;
           #"M".run.PF[#c].%X1 := #"M".readMsgSlot[#c].cmdRespons.FP_2;
           #"M".run.PF[#c].%X2 := #"M".readMsgSlot[#c].cmdRespons.FP_3;
           #"M".run.PF[#c].%X3 := #"M".readMsgSlot[#c].cmdRespons.FP_4;
           #"M".run.PF[#c].%X4 := #"M".readMsgSlot[#c].cmdRespons.FP_5;

           #"M".run.cmdAck[#c].%X0 := #"M".readMsgSlot[#c].cmdRespons.cmdAck1;
           #"M".run.cmdAck[#c].%X1 := #"M".readMsgSlot[#c].cmdRespons.cmdAck2;
       END_FOR;
   END_REGION


   #loadTargetValue(M := #"M",
                    sb := #sb);




   #"M".queryDone.write := false;
   #"M".queryDone.read := false;
END_FUNCTION_BLOCK

FUNCTION "releaseMsgSlot" : Void   // FC17, SCL
{ S7_Optimized_Access := 'TRUE' }
VERSION : 0.1
   VAR_IN_OUT
      slot : USInt;
      mem : Array[*] of Bool;
   END_VAR
   VAR_TEMP
      c : Int;
   END_VAR
BEGIN

   IF #slot <> 0 THEN
       #mem[#slot] := false;
   END_IF;
END_FUNCTION

FUNCTION "reqMsgSlot" : USInt   // FC18, SCL
{ S7_Optimized_Access := 'TRUE' }
VERSION : 0.1
   VAR_IN_OUT
      mem : Array[*] of Bool;
   END_VAR
   VAR_TEMP
      c : Int;
   END_VAR
BEGIN
   // Find first entry inside mem that is false.
   // set the entry to true and return the index. 

   #reqMsgSlot := 0;
   FOR #c := LOWER_BOUND(ARR := #mem, DIM := 1) TO
       UPPER_BOUND(ARR := #mem, DIM := 1)
   DO
       IF NOT #mem[#c] THEN
           #mem[#c] := true;
           #reqMsgSlot := INT_TO_USINT(#c);
           RETURN;
       END_IF;
   END_FOR;
END_FUNCTION

// folder: Library/Modbus/Station blocks/sb untested/Produal

FUNCTION_BLOCK "produal_KLH_M"   // FB42, SCL
{ S7_Optimized_Access := 'TRUE' }
VERSION : 0.1
   VAR_INPUT
      mb_addr : USInt;
   END_VAR
   VAR_OUTPUT
      temperature : Real;
      humidity : Real;
      potentiometer : Real;
   END_VAR
   VAR_IN_OUT
      mb_query : "mb_query";
   END_VAR
   VAR
      sb : "mb_station_block_udt";
      write1_calibration : Struct
         temp_offset : Int;
         humidity_offset : Int;
      END_STRUCT;
      read1 : Struct
         temperature : Int;
         humidity : UInt;
         y : Array[1..4] of UInt;
         potentiometer : Int;   // %
      END_STRUCT;
   END_VAR
BEGIN
   // Produal - KLH-M
   // Product number: 1132600
   // http://www.produal.com/shop/web_humidity_transmitters/sku-1132600

   "mb_station_block_header"(sb := #sb, mb_query := #mb_query);
   #mb_query.mb_addr := #mb_addr;

   #mb_query(mode := #mb_query.c.mode.read,
             data_addr := 30001,
             data_ptr := #read1);

   #mb_query(mode := #mb_query.c.mode.write,
             data_addr := 40006,
             data_ptr := #write1_calibration); // temp. and humidity  

   "mb_station_block_footer"(sb := #sb, mb_query := #mb_query);

   #temperature := INT_TO_REAL(#read1.temperature) * 0.1;
   #humidity := UINT_TO_REAL(#read1.humidity); // 0-100%
   #potentiometer := INT_TO_REAL(#read1.potentiometer) * 0.1;
END_FUNCTION_BLOCK

FUNCTION_BLOCK "produal_TEHR_M"   // FB43, SCL
{ S7_Optimized_Access := 'TRUE' }
VERSION : 0.1
   VAR_INPUT
      mb_addr : USInt;
      calibration_offset : Int;   // mbar
   END_VAR
   VAR_OUTPUT
      temperature : Real;   // Â°C
      analogue_output : Real;   // V
      potentiometer : Real;   // %
   END_VAR
   VAR_IN_OUT
      mb_query : "mb_query";
   END_VAR
   VAR
      sb : "mb_station_block_udt";
      r1 : Struct
         temperature : Int;
         analogue_output : UInt;
         potentiometer : Int;
      END_STRUCT;
   END_VAR
BEGIN
   // Produal - TEHR-M - Temperatur transmitter.
   // Product: 117Z190 - Pt1000 EN 60751/B
   // http://www.produal.com/shop/web_bus_temperature_transmitters/
   // sku-117Z190?hiddenAttributes_sensor_output=sensor_output_modbus&saf=true

   "mb_station_block_header"(sb := #sb,
                             mb_query := #mb_query);
   #mb_query.mb_addr := #mb_addr;

   #mb_query(mode := #mb_query.c.mode.read,
             data_addr := 30001,
             data_ptr := #r1);

   #mb_query(mode := #mb_query.c.mode.write,
             data_addr := 40001,
             data_ptr := #calibration_offset);

   "mb_station_block_footer"(sb := #sb,
                             mb_query := #mb_query);

   #temperature := INT_TO_REAL(#r1.temperature) * 0.1;
   #analogue_output := UINT_TO_REAL(#r1.analogue_output);
   #potentiometer := INT_TO_REAL(#r1.potentiometer) * 0.1;
END_FUNCTION_BLOCK

// folder: Library/Modbus/Station blocks/sb untested/Scandinavian Electric

FUNCTION_BLOCK "Scandinavian_electric_CEM M-RS485"   // FB45, SCL
{ S7_Optimized_Access := 'TRUE' }
VERSION : 0.1
   VAR_INPUT
      mb_addr : UInt;
   END_VAR
   VAR_IN_OUT
      mb_query : "mb_query";
   END_VAR
   VAR
      sb : "mb_station_block_udt";
      read1 : Struct
         "Imported active energy" : UDInt;
         "Exported active energy" : UDInt;
         "Q1 Reactive energy" : UDInt;
         "Q2 Reactive energy" : UDInt;
         "Q3 Reactive energy" : UDInt;
         "Q4 Reactive energy" : UDInt;
      END_STRUCT;
      read2 : Struct
         "Partial imported active energy" : UDInt;
         "Partial exported active energy" : UDInt;
         "Q1 partial reactive energy" : UDInt;
         "Q2 partial reactive energy" : UDInt;
         "Q3 partial reactive energy" : UDInt;
         "Q4 partial reactive energy" : UDInt;
      END_STRUCT;
      serial_number : UDInt;
   END_VAR
BEGIN
   // Scandinavian Electric - Circutor - CEM M-RS485
   // Modbus interface for CEM energy meters

   // - Note: Only no parity.
   // - http://scel.no/produkter/energimaling_/_3_fase_malere/
   //   content/text_432575b2-b97f-4834-84d7-3fb83a2fdd40/1442214133237/
   //   cem_m_rs485.pdf
   // - (M014B01-03-14A)

   "mb_station_block_header"(sb := #sb, mb_query := #mb_query);
   #mb_query.mb_addr := #mb_addr;

   #mb_query.mode := #mb_query.c.read.holding_reg;
   #mb_query(data_addr := 16#0000, data_ptr := #read1);
   #mb_query(data_addr := 16#0030, data_ptr := #read2);
   #mb_query(data_addr := 16#2710, data_ptr := #serial_number);

   "mb_station_block_footer"(sb := #sb, mb_query := #mb_query);
END_FUNCTION_BLOCK

FUNCTION_BLOCK "Scandinavian_electric_Circutor_CBS"   // FB46, SCL
{ S7_Optimized_Access := 'TRUE' }
VERSION : 0.1
   VAR_INPUT
      mb_addr : UInt;
   END_VAR
   VAR_IN_OUT
      mb_query : "mb_query";
   END_VAR
   VAR
      sb : "mb_station_block_udt";
      data : Struct
         current : Array[1..8] of UInt;   // [mA]
         outputs : Array[1..8] of UInt;   // 0=Normal, 1=Pre-alarm, 2=Aktivert, 3=LÃ¥st
         pre_alarm_relay : UInt;
      END_STRUCT;
      limits : Array[1..8] of UInt;   // [mA]
   END_VAR
BEGIN
   // Scandinavian Electric - Circutor - CBS-8
   // 
   // - http://scel.no/produkter/jordfeilovervaking/
   //   varsler_panel_og_scanningsystem/content_2/
   //   text_8e3609e0-231d-4dfc-80a4-71ee43eee1af/1409662445698/cbs8.pdf

   "mb_station_block_header"(sb := #sb, mb_query := #mb_query);
   #mb_query.mb_addr := #mb_addr;

   #mb_query.mode := #mb_query.c.write.holding_reg;
   #mb_query(data_addr := 13, data_ptr := #limits);

   #mb_query.mode := #mb_query.c.read.holding_reg;
   #mb_query(data_addr := 2, data_ptr := #data);

   "mb_station_block_footer"(sb := #sb, mb_query := #mb_query);
END_FUNCTION_BLOCK

// folder: Library/Modbus/Station blocks/sb untested/Schneider

FUNCTION_BLOCK "Schneider_ATV6xx"   // FB47, SCL
{ S7_Optimized_Access := 'TRUE' }
VERSION : 0.1
   VAR_INPUT
      mb_addr : USInt;
      ref_freq : Real;
   END_VAR
   VAR_IN_OUT
      mb_query : "mb_query";
   END_VAR
   VAR
      sb : "mb_station_block_udt";
      write1 : Struct
         cmd_reg : Struct
            x08_halt : Bool;
            x09 : Bool;
            x10 : Bool;
            x11_Reverse : Bool;
            x12 : Bool;
            x13 : Bool;
            x14 : Bool;
            x15 : Bool;
            x00_switch_on : Bool := TRUE;
            x01_enable_voltage : Bool := TRUE;
            x02_quick_stop : Bool;
            x03_Run : Bool;
            x04 : Bool;
            x05 : Bool;
            x06 : Bool;
            x07_fault_reset : Bool;
         END_STRUCT;
         ref_freq : Int;
      END_STRUCT;
      read1 : Struct
         status : Struct   // ETA
            x08 : Bool;
            x09_remote : Bool;   // Command or reference value via fieldbus
            x10_on_target : Bool;   // Reference value reached
            x11_ref_outside_lim : Bool;   // Reference value outside limits
            x12 : Bool;
            x13 : Bool;
            x14_stop_key : Bool;   // Manufacturer-specific Stop via STOP key
            x15_reverse : Bool;   // Manufacturer-specific
            x00_awaiting_power_stage_supply : Bool;
            x01_ready : Bool;
            x02_running : Bool;
            x03_fault : Bool;
            x04_power_stage_supply_present : Bool;
            x05_quick_stop : Bool;
            x06_power_stage_supply_disabled : Bool;
            x07_warning : Bool;
         END_STRUCT;
         output_frequency : Int;   // RFR
         frequency_reference_before_ramp : Int;   // FRH
         motor_current : Int;   // LCR
         motor_torque : Int;   // OTR
         ext_status_word : Word;
         mains_voltage : Int;   // ULN
         motor_voltage : Int;   // UOP
         drive_thermal_state : Int;   // THD
      END_STRUCT;
   END_VAR
BEGIN
   // Schneider - ATV6xx (EAV94279)
   //  
   // - http://www2.schneider-electric.com/resources/sites/SCHNEIDER_ELECTRIC/
   //   content/live/FAQS/275000/FA275868/en_US/
   //   Process%20drive%20communication%20parameters.xlsx
   // - https://profsector.com/media/catalogs/56e3af69500ef.pdf
   // - https://download.schneider-electric.com/
   //   files?p_enDocType=User+guide&p_File_Id=5470508810&
   //   p_File_Name=ATV600_EthernetIP_Modbus_TCP_Manual_EN_EAV6
   //   4328_02.pdf&p_Reference=EAV64328

   #write1.ref_freq := REAL_TO_INT(#ref_freq * 10);
   #write1.cmd_reg.x00_switch_on := #write1.cmd_reg.x03_Run := #ref_freq <> 0;

   "mb_station_block_header"(sb := #sb, mb_query := #mb_query);
   #mb_query.mb_addr := #mb_addr;

   #mb_query.mode := #mb_query.c.write.holding_reg;
   #mb_query(data_addr := 8501, data_ptr := #write1);

   #mb_query.mode := #mb_query.c.read.holding_reg;
   #mb_query(data_addr := 3201, data_ptr := #read1);

   "mb_station_block_footer"(sb := #sb, mb_query := #mb_query);
END_FUNCTION_BLOCK

FUNCTION_BLOCK "Schneider_PM556x_series"   // FB48, SCL
{ S7_Optimized_Access := 'TRUE' }
VERSION : 0.1
   VAR_INPUT
      mb_addr : UInt;
   END_VAR
   VAR_IN_OUT
      mb_query : "mb_query";
   END_VAR
   VAR
      sb : "mb_station_block_udt";
      Accumulated_Energy : Struct
         "Active Energy Delivered (Into Load)" : Real;   // kWh
         "Active Energy Received (Out of Load)" : Real;   // kWh
         "Active Energy Delivered + Received" : Real;   // kWh
         "Active Energy Delivered- Received" : Real;   // kWh
         "Reactive Energy Delivered" : Real;   // kVARh
         "Reactive Energy Received" : Real;   // kVARh
         "Reactive Energy Delivered + Received" : Real;   // kVARh
         "Reactive Energy Delivered - Received" : Real;   // kVARh
         "Apparent Energy Delivered" : Real;   // kVAh
         "Apparent Energy Received" : Real;   // kVAh
         "Apparent Energy Delivered + Received" : Real;   // kVAh
         "Apparent Energy Delivered - Received" : Real;   // kVAh
      END_STRUCT;
      data1 : Struct
         Current : Array[1..3] of Real;   // A
         "Current N" : Real;   // A
         "Current G" : Real;   // A
         "Current Avg" : Real;   // A
         "Current Unbalance" : Array[1..3] of Real;   // %
         "Current Unbalance Worst" : Real;   // %
         "Voltage L-L" : Array[1..3] of Real;   // V
         "Voltage L-L Avg" : Real;   // V
         "Voltage L-N" : Array[1..3] of Real;   // V
         "Voltage L-N Avg" : Real;   // V
         "Voltage Unbalance L-L" : Array[1..3] of Real;   // %
         "Voltage Unbalance L-L Worst" : Real;   // %
         "Voltage Unbalance L-N" : Array[1..3] of Real;   // %
         "Voltage Unbalance L-N Worst" : Real;   // %
      END_STRUCT;
      Power : Struct
         "Active Power" : Array[1..3] of Real;   // kW
         "Active Power Total" : Real;   // kW
         "Reactive Power" : Array[1..3] of Real;   // kVAR
         "Reactive Power Total" : Real;   // kVAR
         "Apparent Power" : Array[1..3] of Real;   // kVA
         "Apparent Power Total" : Real;   // kVA
         "Power Factor" : Array[1..3] of Real;   // ---
         "Power Factor Total" : Real;   // ---
         "Displacement Power Factor" : Array[1..3] of Real;   // ---
         "Displacement Power Factor Total" : Real;   // ---
      END_STRUCT;
      PF : Struct
         "Power Factor" : Array[1..3] of Real;
         "Power Factor Total" : Real;
         "Displacement Power Factor" : Array[1..3] of Real;
         "Displacement Power Factor Total" : Real;
      END_STRUCT;
      Frequency : Real;   // Hz
   END_VAR
   VAR_TEMP
      c : Int;
      t1 : Real;
      t2 : Real;
   END_VAR
BEGIN
   // Schneider Electric - PM5560, PM5563, PM5563RD
   // 
   // https://www.schneider-electric.com/en/faqs/FA234017/

   "mb_station_block_header"(sb := #sb, mb_query := #mb_query);
   #mb_query.mb_addr := #mb_addr;

   #mb_query.mode := #mb_query.c.read.holding_reg;
   #mb_query(data_addr := 2700, data_ptr := #Accumulated_Energy);
   #mb_query(data_addr := 3000, data_ptr := #data1);
   #mb_query(data_addr := 3054, data_ptr := #Power);
   #mb_query(data_addr := 3110, data_ptr := #Frequency);

   "mb_station_block_footer"(sb := #sb, mb_query := #mb_query);

   FOR #c := 1 TO 8 DO
       (* Power factor values are specially encoded floating point 
       values. Angle of complex power = power factor register value
       0° = 1, 90° = 0,  180° = -1,  270° = 2,  Q1: 0 < x < 1
       Q2: -2 < x < -1,  Q3:  -1 < x < 0,   Q4: 1 < x < 2  *)
       CASE #c OF
           1..3: #t1 := #Power."Power Factor"[#c];
           4:    #t1 := #Power."Power Factor Total";
           5..7: #t1 := #Power."Displacement Power Factor"[#c - 4];
           8:    #t1 := #Power."Displacement Power Factor Total";
       END_CASE;
       IF #t1 > 1 THEN // PF is leading
           #t2 := 2 - #t1;
       ELSIF #t1 < -1 THEN // PF is leading
           #t2 := -2 - #t1;
       ELSE            // ABS(#t1) = 1 -> PF is at unity
           #t2 := #t1; // else -> PF is lagging
       END_IF;
       CASE #c OF
           1..3: #PF."Power Factor"[#c] := #t2;
           4:    #PF."Power Factor Total" := #t2;
           5..7: #PF."Displacement Power Factor"[#c - 4] := #t2;
           8:    #PF."Displacement Power Factor Total" := #t2;
       END_CASE;
   END_FOR;
END_FUNCTION_BLOCK

FUNCTION_BLOCK "Schneider_PM1000_series"   // FB49, SCL
TITLE = Schneider Electric - PM1000 Series Power Meters
{ S7_Optimized_Access := 'TRUE' }
VERSION : 0.1
   VAR_INPUT
      mb_addr : UInt;
   END_VAR
   VAR_OUTPUT
      all : Struct
         apparent_power : Real;
         active_power : Real;
         reactive_power : Real;
         power_factor : Real;
         voltage_L_L : Real;
         voltage_L_N : Real;
         current : Real;
      END_STRUCT;
      phase : Array[1..3] of Struct
         apparent_power : Real;
         active_power : Real;
         reactive_power : Real;
         power_factor : Real;
         voltage_L_L : Real;
         voltage_L_N : Real;
         current : Real;
      END_STRUCT;
   END_VAR
   VAR_IN_OUT
      mb_query : "mb_query";
   END_VAR
   VAR
      sb : "mb_station_block_udt";
   END_VAR
   VAR_TEMP
      tAll : Struct
         apparent_power : DWord;
         active_power : DWord;
         reactive_power : DWord;
         power_factor : DWord;
         voltage_L_L : DWord;
         voltage_L_N : DWord;
         current : DWord;
      END_STRUCT;
      tPhase : Array[1..3] of Struct
         apparent_power : DWord;
         active_power : DWord;
         reactive_power : DWord;
         power_factor : DWord;
         voltage_L_L : DWord;
         voltage_L_N : DWord;
         current : DWord;
      END_STRUCT;
      c : Int;
   END_VAR
BEGIN
   // Schneider Electric - PowerLogic - PM1000 Series Power Meters
   //  - PM1200
   // 
   // http://static.schneider-electric.us/docs/Power%20Management/
   // PowerLogic%20Products/Metering/PM1200%20power%20meter/
   // PLSED309039EN_PM1000_UG.pdf

   "mb_station_block_header"(sb := #sb,
                             mb_query := #mb_query);
   #mb_query.mb_addr := #mb_addr;

   #mb_query.mode := #mb_query.c.read.holding_reg;

   #mb_query(data_addr := 3901,
             data_ptr := #tAll);
   IF #mb_query.Done THEN
       #all.apparent_power := DWORD_TO_REAL(SWAP(#tAll.apparent_power));
       #all.active_power := DWORD_TO_REAL(SWAP(#tAll.active_power));
       #all.reactive_power := DWORD_TO_REAL(SWAP(#tAll.reactive_power));
       #all.power_factor := DWORD_TO_REAL(SWAP(#tAll.power_factor));
       #all.voltage_L_L := DWORD_TO_REAL(SWAP(#tAll.voltage_L_L));
       #all.voltage_L_N := DWORD_TO_REAL(SWAP(#tAll.voltage_L_N));
       #all.current := DWORD_TO_REAL(SWAP(#tAll.current));
   END_IF;

   FOR #c := 1 TO 3 DO
       CASE #c OF
           1:
               #mb_query.data_addr := 3917;
           2:
               #mb_query.data_addr := 3931;
           3:
               #mb_query.data_addr := 3945;
       END_CASE;
       #mb_query(data_ptr := #tPhase[#c]);
       IF #mb_query.Done THEN
           #phase[#c].apparent_power := DWORD_TO_REAL(SWAP(#tPhase[#c].apparent_power));
           #phase[#c].active_power := DWORD_TO_REAL(SWAP(#tPhase[#c].active_power));
           #phase[#c].reactive_power := DWORD_TO_REAL(SWAP(#tPhase[#c].reactive_power));
           #phase[#c].power_factor := DWORD_TO_REAL(SWAP(#tPhase[#c].power_factor));
           #phase[#c].voltage_L_L := DWORD_TO_REAL(SWAP(#tPhase[#c].voltage_L_L));
           #phase[#c].voltage_L_N := DWORD_TO_REAL(SWAP(#tPhase[#c].voltage_L_N));
           #phase[#c].current := DWORD_TO_REAL(SWAP(#tPhase[#c].current));
       END_IF;
   END_FOR;

   "mb_station_block_footer"(sb := #sb,
                             mb_query := #mb_query);
END_FUNCTION_BLOCK

FUNCTION_BLOCK "Schneider_power_meter_750"   // FB50, SCL
{ S7_Optimized_Access := 'TRUE' }
VERSION : 0.1
   VAR_INPUT
      mb_addr : UInt;
   END_VAR
   VAR_IN_OUT
      mb_query : "mb_query";
   END_VAR
   VAR
      sb : "mb_station_block_udt";
      data1 : Struct
         "Real Energy, Total" : Real;   // kWh
         "Apparent Energy,Tota" : Real;   // kVAh
         "Reactive Energy,Tota" : Real;   // kVARh
         "Real Power, Total" : Real;   // kW
         "Apparent Power, Total" : Real;   // kVA
         "Reactive Power, Total" : Real;   // kVAR
         "Power Factor, Total" : Real;
         "Voltage, L-L, 3PAverage" : Real;   // Volt
         "Voltage, L-N, 3PAverage" : Real;   // Volt
         "Current, 3P Average" : Real;   // Amp
         Frequency : Real;
      END_STRUCT;
      data2 : Struct
         Current : Array[1..3] of Real;
         Current_N : Real;
      END_STRUCT;
      data3 : Struct
         Voltage_L_L : Array[1..3] of Real;   // [V] 1:L1-L2, 2:L2-L3, 3:L3-L1
         Voltage_L_N : Array[1..3] of Real;   // [V]
         "Real Power" : Array[1..3] of Real;   // kW
         "Apparent Power" : Array[1..3] of Real;   // kVA
         "Reactive Power" : Array[1..3] of Real;   // kVAR
      END_STRUCT;
   END_VAR
BEGIN
   // Schneider - Power Meter 750
   // 63230-507-201A1 - 03/2007
   // 
   // Web: https://www.ccontrols.com/support/dp/SchneiderElectricPowerMeter750.pdf

   "mb_station_block_header"(sb := #sb,
                             mb_query := #mb_query);
   #mb_query.mb_addr := #mb_addr;

   #mb_query.mode := #mb_query.c.read.holding_reg;
   #mb_query(data_addr := 1000,
             data_ptr := #data1);
   #mb_query(data_addr := 1034,
             data_ptr := #data2);
   #mb_query(data_addr := 1054,
             data_ptr := #data3);

   "mb_station_block_footer"(sb := #sb,
                             mb_query := #mb_query);
END_FUNCTION_BLOCK

FUNCTION_BLOCK "Schneider_SCADAPack_4000"   // FB51, SCL
{ S7_Optimized_Access := 'TRUE' }
VERSION : 0.1
   VAR_INPUT
      mb_addr : UInt;
   END_VAR
   VAR_IN_OUT
      mb_query : "mb_query";
   END_VAR
   VAR
      sb : "mb_station_block_udt";
      data : Array[1..3] of Int;
      setting : Array[1..3] of Int;
   END_VAR
BEGIN
   // Schneider - SCADAPack 4000 
   // Models 4012, 4032 and 4102 - Transmitters
   // 
   // Web: https://s3.amazonaws.com/cdn.freshdesk.com/data/helpdesk/
   // attachments/production/5013914262/original/
   // SCADAPack_4000_Series_Transmitters.pdf?
   // X-Amz-Algorithm=AWS4-HMAC-SHA256&X-Amz-Credential=
   // AKIAJ2JSYZ7O3I4JO6DA%2F20170919%2Fus-east-1%2Fs3%2Faws4_
   // request&X-Amz-Date=20170919T163931Z&X-Amz-Expires=300&X-Amz-
   // Signature=a206005821114e23f4a38162afdf9d14bd82209c246a378f18
   // 9af628740a1509&X-Amz-SignedHeaders=Host&response-content-type=
   // application%2Fpdf

   "mb_station_block_header"(sb := #sb, mb_query := #mb_query);
   #mb_query.mb_addr := #mb_addr;

   #mb_query.mode := #mb_query.c.mode.read;
   #mb_query(data_addr := 40116, data_ptr := #data);

   #mb_query.mode := #mb_query.c.mode.write;
   #mb_query(data_addr := 40060, data_ptr := #setting);

   "mb_station_block_footer"(sb := #sb, mb_query := #mb_query);

   (*
   Setting:

   value[1] and value[2]
   ------------------
   2 = Pascal (Pa)
   3 = kiloPascal (kPa)
   4 = megaPascal (MPa)
   5 = pounds per square inch (psi)
   6 = inches of water at 68 F
   7 = ftH2O
   8 = atm
   9 = bar
   10 = kg/cm2
   11 = g/cm2
   12 = cmHg
   13 = mmHg
   14 = torr
   15 = mH2O
   16 = cmH2O
   17 = mmH2O
   18 = inHg
   19 = mbar


   value[3]
   ------------------
   20 = degrees Celsius (ï‚°C)
   21 = degrees Fahrenheit (ï‚°F)
   22 = degrees Kelvin (K)
   23 = degrees Rankine(R)

   *)
END_FUNCTION_BLOCK

FUNCTION_BLOCK "Schneider_conzerv_EM6430"   // FB91, SCL
{ S7_Optimized_Access := 'TRUE' }
VERSION : 0.1
   VAR_INPUT
      mb_addr : USInt;
   END_VAR
   VAR_IN_OUT
      mb_query : "mb_query";
   END_VAR
   VAR
      sb : "mb_station_block_udt";
      read1_common : Struct
         Apparent_power_total : Real;
         Active_power_total : Real;
         Reactive_power_total : Real;
         Power_factor_average : Real;
         Voltage_average_phase_phase : Real;
         Voltage_average_phase_neutral : Real;
         Current_average : Real;
         Frequency : Real;   // Hz
      END_STRUCT;
      read2_phase : Array[1..3] of Struct
         Apparent_power : Real;
         Active_power : Real;
         Reactive_power : Real;
         Power_factor : Real;
         Voltage_phase_phase : Real;
         Voltage_phase_neutral : Real;
         Current : Real;
      END_STRUCT;
      read3_THD : Struct
         Voltage_THD : Array[1..3] of Real;
         Current_THD : Array[1..3] of Real;
      END_STRUCT;
      read4 : Struct
         Forward_apparent_energy : Real;
         Forward_active_energy : Real;
         Forward_reactive_inductive_energy : Real;
         Forward_reactive_capacitive_energy : Real;
         Reverse_apparent_energy : Real;
         Reverse_active_energy : Real;
         Reverse_reactive_inductive_Energy : Real;
         Reverse_reactive_capacitive_Energy : Real;
         Average_load_percentage : Real;
         Percentage_of_phase_load : Array[1..3] of Real;
         "Unbalanced_%load" : Real;
         "Unbalanced_%_voltage" : Real;
      END_STRUCT;
      read5_common_RMS : Struct
         Apparent_power_total : Real;
         Active_power_total : Real;
         Reactive_power_total : Real;
         Power_factor_average : Real;
         Voltage_average_phase_phase : Real;
         Voltage_average_phase_neutral : Real;
         Current_average : Real;
         Frequency : Real;   // Hz
         _ : UDInt;   // Reserved
         Number_of_interruption : UDInt;
      END_STRUCT;
   END_VAR
BEGIN
   // Schneider-electric - Conzerv EM6430 - Power meters
   // NHA12535-03
   // 
   // https://www.schneider-electric.com/resources/sites/SCHNEIDER_ELECTRIC/
   // content/live/FAQS/276000/FA276938/en_US/EM6430_User_Manual_NHA12535-03.pdf

   "mb_station_block_header"(sb := #sb, mb_query := #mb_query);
   #mb_query.mb_addr := #mb_addr; // Device address.

   #mb_query.mode := #mb_query.c.read.holding_reg;
   #mb_query(data_addr := 3901, data_ptr := #read1_common);
   #mb_query(data_addr := 3917, data_ptr := #read2_phase);
   #mb_query(data_addr := 3861, data_ptr := #read3_THD);
   #mb_query(data_addr := 3959, data_ptr := #read4);
   #mb_query(data_addr := 3001, data_ptr := #read5_common_RMS);

   "mb_station_block_footer"(sb := #sb, mb_query := #mb_query);
END_FUNCTION_BLOCK

FUNCTION_BLOCK "Schneider_PM750"   // FB92, SCL
{ S7_Optimized_Access := 'TRUE' }
VERSION : 0.1
   VAR_INPUT
      mb_addr : UInt;
   END_VAR
   VAR_IN_OUT
      mb_query : "mb_query";
   END_VAR
   VAR
      sb : "mb_station_block_udt";
      data1 : Struct
         "Real Energy, Total" : Real;   // kWh
         "Apparent Energy,Tota" : Real;   // kVAh
         "Reactive Energy,Tota" : Real;   // kVARh
         "Real Power, Total" : Real;   // kW
         "Apparent Power, Total" : Real;   // kVA
         "Reactive Power, Total" : Real;   // kVAR
         "Power Factor, Total" : Real;
         "Voltage, L-L, 3PAverage" : Real;   // Volt
         "Voltage, L-N, 3PAverage" : Real;   // Volt
         "Current, 3P Average" : Real;   // Amp
         Frequency : Real;
      END_STRUCT;
      data2 : Struct
         Current : Array[1..3] of Real;
         Current_N : Real;
      END_STRUCT;
      data3 : Struct
         Voltage_L_L : Array[1..3] of Real;   // [V] 1:L1-L2, 2:L2-L3, 3:L3-L1
         Voltage_L_N : Array[1..3] of Real;   // [V]
         "Real Power" : Array[1..3] of Real;   // kW
         "Apparent Power" : Array[1..3] of Real;   // kVA
         "Reactive Power" : Array[1..3] of Real;   // kVAR
      END_STRUCT;
   END_VAR
BEGIN
   // Schneider - Power Meter 750
   // 63230-507-201A1 - 03/2007
   // 
   // Web: https://www.ccontrols.com/support/dp/SchneiderElectricPowerMeter750.pdf

   "mb_station_block_header"(sb := #sb, mb_query := #mb_query);
   #mb_query.mb_addr := #mb_addr;

   #mb_query.mode := #mb_query.c.read.holding_reg;
   #mb_query(data_addr := 1000, data_ptr := #data1);
   #mb_query(data_addr := 1034, data_ptr := #data2);
   #mb_query(data_addr := 1054, data_ptr := #data3);

   "mb_station_block_footer"(sb := #sb, mb_query := #mb_query);
END_FUNCTION_BLOCK

FUNCTION_BLOCK "Schneider_Altivar_21"   // FB95, SCL
{ S7_Optimized_Access := 'TRUE' }
VERSION : 0.1
   VAR_INPUT
      mb_addr : UInt;
      ref : Real;
      acceleration_time : Real;
   END_VAR
   VAR_IN_OUT
      mb_query : "mb_query";
   END_VAR
   VAR
      sb : "mb_station_block_udt";
      data6 : Struct
         Output_current : Real;
         Voltage_DC_bus : Real;
         Output_frequency : Real;
      END_STRUCT;
      read1 : Struct   // 16#fd00
         Output_frequency : Word;
         stat : Struct
            x08 : Bool;
            x09_Reverse : Bool;
            x10_Run : Bool;
            x11_Coast_stop : Bool;
            x12_Emergency_stop : Bool;
            x13_Standby_ST_ON : Bool;   // Standby: Initialization completed, not failure stop status, not alarm stop status (MOFF, LL forced stop or forced stop due to a momentary power failure), ST=ON, and RUN=ON
            x14_Standby : Bool;   // Standby: Initialization completed, not failure stop status, and not alarm stop status (MOFF, LL forced stop or forced stop due to a momentary power failure)
            x15_Local : Bool;
            x00_Failure_FL : Bool;
            x01_Failure : Bool;
            x02_Alarm : Bool;
            x03_Main_circuit_undervoltage : Bool;
            x04_THR_2 : Bool;   // THR1: PT=set value, vL, vb, Thr - THR2: PT=0, F170, F172, F173
            x05_PI_control_OFF : Bool;
            x06_Acceleration2_deceleration2 : Bool;
            x07_DC_braking : Bool;
         END_STRUCT;
      END_STRUCT;
      read2 : Struct   // 16#fe45
         Command_mode : UInt;   // 0:Terminal board, 1:Operation panel, 2:Serial
         Setpoint_mode : UInt;   // 1 VIA, 2 VIB, 3 Operation panel, 4 Serial, 5 TB up down frequency, 255 Preset speed operation
      END_STRUCT;
      read3_alarm : Struct   // 16#fe91
         x08_Over_torque : Bool;
         x09_Cumulative_operation_hours : Bool;
         x10 : Bool;
         x11 : Bool;
         x12 : Bool;
         "x13_Main circuit_undervoltage" : Bool;   // same as MS-relay status
         x14_Decelerating_stopping : Bool;   // Related: F256 setting. At the time of the instant blackout, Forced deceleration/stop
         x15_Decelerating_stopping : Bool;   // Related: F302 setting. An automatic stop during the lower limit frequency continuance
         x00_Overcurrent : Bool;
         x01_Inverter_overload : Bool;
         x02_Motor_overload : Bool;
         x03_Overheat : Bool;
         x04_Overvoltage : Bool;
         x05_Main_circuit_undervoltage : Bool;
         x06 : Bool;
         x07_Undercurrent : Bool;
      END_STRUCT;
      read4_alarm2 : Struct   // 16#fe79
         x08 : Bool;
         x09 : Bool;
         x10 : Bool;
         x11 : Bool;
         x12 : Bool;
         x13 : Bool;
         x14 : Bool;
         x15 : Bool;
         x00_Fan_life_alarm : Bool;
         x01_Circuit_board_life : Bool;
         x02_Main_circuit_capacitor_life : Bool;
         x03_User_set_alarm : Bool;
         x04 : Bool;
         x05 : Bool;
         x06 : Bool;
         x07 : Bool;
      END_STRUCT;
      read5_trip_code : UInt;   // 16#fc90
      write1 : Struct
         cmd : Struct
            x08 : Bool;   // [08]
            reverse : Bool;   // [09]
            run : Bool;   // [10]
            coast_stop : Bool;   // [11]
            emergency_stop : Bool;   // [12]
            fault_reset : Bool;   // [13]
            setpoint_priority : Bool := TRUE;   // [14] Enabled regardless of the setting of FMOD
            command_priority : Bool := TRUE;   // [15] Enabled regardless of the setting of CMOD
            preset_speed_b0 : Bool;   // [00]
            preset_speed_b1 : Bool;   // [01]
            preset_speed_b2 : Bool;   // [02]
            x03 : Bool;   // [03]
            thr2 : Bool;   // [04] THR1 : PT=set value, vL, vb, tHr - THR2 : PT=0, F170, F172, F173
            PI_control : Bool;   // [05] 0:Normal operation, 1:PI OFF
            acceleration_deceleration_pattern_2 : Bool;   // [06] 0: Acceleration deceleration pattern 1
            DC_braking : Bool;   // [07]
         END_STRUCT;
         ref : UInt;
      END_STRUCT;
      write2_comm_fault_action : UInt;
      _ : Bool;
      sequence : "mb_sequence";
   END_VAR
   VAR_TEMP
      read6 : Struct   // 16#fe03
         Output_current : UInt;
         Voltage_DC_bus : UInt;
      END_STRUCT;
      u : UInt;
   END_VAR
BEGIN
   // Schneider (Telemecanique) - Altivar 21 inverter
   // VFD (AC-drive)

   (*
   Param:  Name:             Default:    Options:          
   F800    Baud rate         19200       0: 9600 bps, 1: 19200 bps     
   F801    Parity            Even        0: None, 1: Even, 2: Odd      
   F802    Modbus address    1           0 ... 247                     

   CMOD    2 -> Serial communication
   FMOD    4 -> Serial communication
   *)

   "mb_station_block_header"(sb := #sb, mb_query := #mb_query);
   #mb_query.mb_addr := #mb_addr;

   REGION Low priority queries     
       #sequence.conf.first_state := 1600;
       CASE "mb_sequence_init"(sequence := #sequence, mb_query := #mb_query) OF
               // ----- READ HOLDING REG ----- (State 3xx)
           300: // Where the drive take commands from: modbus or Terminal board.
               #mb_query(data_addr := 16#fe45, data_ptr := #read2); // 65093
           301: #mb_query(data_addr := 16#fe91, data_ptr := #read3_alarm);
           302: #mb_query(data_addr := 16#fe79, data_ptr := #read4_alarm2);
           303: #mb_query(data_addr := 16#fc90, data_ptr := #read5_trip_code);
           304: // Other data: Current, DC-bus
               #mb_query(data_addr := 16#fe03, data_ptr := #read6);
               IF #mb_query.Done THEN
                   #data6.Output_current := UINT_TO_REAL(#read6.Output_current) / 100;
                   #data6.Voltage_DC_bus := UINT_TO_REAL(#read6.Voltage_DC_bus) / 100;
               END_IF;
               #sequence.next_state := 1600;

               // ----- WRITE MULTIPLE HOLDING REG ----- (State 16xx)
           1600: // Behaviour on modbus fault
               #mb_query(data_addr := 16#f603, data_ptr := #write2_comm_fault_action);
           1601: // Acceleration time 1  (0.1)
               #u := REAL_TO_UINT(#acceleration_time * 10);
               #mb_query(data_addr := 16#f603, data_ptr := #u);
               #sequence.next_state := 300;
           ELSE
               #sequence.state += 1;
       END_CASE;
       #sequence(sb := #sb, mb_query := #mb_query);
   END_REGION

   REGION High priotiry querie   

       #write1.ref := REAL_TO_UINT(#ref * 100);
       #write1.cmd.run := #ref <> 0 AND #sequence.Done;
       #mb_query(mode := #mb_query.c.write.holding_reg, // 64000
                 data_addr := 16#fa00,
                 data_ptr := #write1);

       // Basic data, status word.
       #mb_query(mode := #mb_query.c.read.holding_reg,
                 data_addr := 16#fd00,
                 data_ptr := #read1); // 64768
       IF #mb_query.Done THEN
           #data6.Output_frequency :=
           (* *)UINT_TO_REAL(#read1.Output_frequency) / 100; // [%]
       END_IF;
   END_REGION

   "mb_station_block_footer"(sb := #sb, mb_query := #mb_query);

   (* Trip codes:
   NErr     0  0  No error
   OC1      1  1  Over-current during acceleration
   OC2      2  2  Over-current during deceleration
   OC3      3  3  Over-current during constant speed operation
   OCL      4  4  Over-current in load at startup
   OCA      5  5  Short circuit in arm
   EPHI     8  8  Input phase failure
   EPHO     9  9  Output phase failure
   OP1      A 10 Overvoltage during acceleration
   OP2      B 11 Overvoltage during deceleration
   OP3      C 12 Overvoltage during constant speed operation
   OL1      D 13 Over-LOAD in inverter
   OL2      E 14 Over-LOAD in motor
   OH      10 16 Overheat trip
   E       11 17 Emergency stop
   EEP1    12 18 EEPROM fault 1 (writing error)
   EEP2    13 19 EEPROM fault 2 (reading error)
   EEP3    14 20 EEPROM fault 3 (internal fault)
   Err2    15 21 RAM fault
   Err3    16 22 ROM fault
   Err4    17 23 CPU fault
   Err5    18 24 Communication error trip
   Err7    1A 26 Current detector fault
   Err8    1B 27 Optional circuit board type error
   UC      1D 29 Small-current trip
   UP1     1E 30 Trip due to undervoltage in main circuit
   Ot      20 32 Over-torque trip
   EF2     22 34 Ground fault trip (hardware detection)
   OC1P    25 37 Overcurrent flowing in element during acceleration
   OC2P    26 38 Overcurrent flowing in element during deceleration
   OC3P    27 39 Overcurrent flowing in element during operation
   EtYP    29 41 Inverter type error
   OH2     2E 46 External thermal input
   SOUt    2F 47 VIA cable break
   E-18    32 50 Break in an analog signal cable
   E-19    33 51 CPU fault
   E-20    34 52 Excess torque boost
   E-21    35 53 CPU fault
   Etn1    54 84 Auto-tuning error
   *)
END_FUNCTION_BLOCK

// folder: Library/Modbus/Station blocks/sb untested/Siemens

FUNCTION_BLOCK "Siemens_7SR11_7SR12_argus"   // FB53, SCL
{ S7_Optimized_Access := 'TRUE' }
VERSION : 0.1
   VAR_INPUT
      mb_addr : USInt := 1;
   END_VAR
   VAR_OUTPUT
      out1 : Struct
         primary_Voltage_L_L : Array[1..3] of Real;
         primary_Voltage_L_N : Array[1..3] of Real;
         secondary_Voltage_L_N : Array[1..3] of Real;
      END_STRUCT;
      out2 : Struct
         nominal_voltage_degrees_L_L : Array[1..3] of Real;
         nominal_voltage_degrees_L_N : Array[1..3] of Real;
         Vzps : Real;
         Vpps : Real;
         Vnps : Real;
         Vzps_degree : Real;
         Vpps_degree : Real;
         Vnps_degree : Real;
         frequency : Real;
      END_STRUCT;
      out3 : Struct
         primary_current : Array[1..3] of Real;
         secondary_current : Array[1..3] of Real;
         nominal_current : Array[1..3] of Real;
         nominal_current_degrees : Array[1..3] of Real;
         primary_In : Real;
         secondary_In : Real;
         nominal_In : Real;
         primary_Ig : Real;
         secondary_Ig : Real;
         nominal_Ig : Real;
         nominal_Izps : Real;
         nominal_Ipps : Real;
         nominal_Inps : Real;
         nominal_Izps_degrees : Real;
         nominal_Ipps_degrees : Real;
         nominal_Inps_degrees : Real;
      END_STRUCT;
      out4 : Struct
         active_power : Array[1..3] of Real;
         active_power_tot : Real;
         reactive_power : Array[1..3] of Real;
         reactive_power_tot : Real;
         apparent_power : Array[1..3] of Real;
         apparent_power_tot : Real;
         power_factor : Array[1..3] of Real;
         power_factor_tot : Real;
      END_STRUCT;
   END_VAR
   VAR_IN_OUT
      mb_query : "mb_query";
   END_VAR
   VAR
      sb : "mb_station_block_udt";
      out5 : Struct
         act_energy_exp : UDInt;
         act_energy_imp : UDInt;
         react_energy_exp : UDInt;
         react_energy_imp : UDInt;
         thermal_status_Ph_A : UInt;
         thermal_status_Ph_B : UInt;
         thermal_Status_Ph_C : UInt;
      END_STRUCT;
      out6 : Struct
         fault_records : Real;
         event_records : Real;
         waveform_records : Real;
         secondary_voltage : Array[1..3] of Real;
      END_STRUCT;
   END_VAR
   VAR_TEMP
      c : Int;
      read1 : Struct
         primary_Voltage_L_L : Array[1..3] of UDInt;
         primary_Voltage_L_N : Array[1..3] of UDInt;
         secondary_Voltage_L_N : Array[1..3] of UDInt;
      END_STRUCT;
      read2 : Struct
         nominal_voltage_degrees_L_L : Array[1..3] of UDInt;
         nominal_voltage_degrees_L_N : Array[1..3] of UDInt;
         Vzps : UDInt;
         Vpps : UDInt;
         Vnps : UDInt;
         Vzps_degree : UDInt;
         Vpps_degree : UDInt;
         Vnps_degree : UDInt;
         frequency : UDInt;
      END_STRUCT;
      read3 : Struct
         primary_current : Array[1..3] of UDInt;
         secondary_current : Array[1..3] of UDInt;
         nominal_current : Array[1..3] of UDInt;
         nominal_current_degrees : Array[1..3] of UDInt;
         primary_In : UDInt;
         secondary_In : UDInt;
         nominal_In : UDInt;
         primary_Ig : UDInt;
         secondary_Ig : UDInt;
         nominal_Ig : UDInt;
         nominal_Izps : UDInt;
         nominal_Ipps : UDInt;
         nominal_Inps : UDInt;
         nominal_Izps_degrees : UDInt;
         nominal_Ipps_degrees : UDInt;
         nominal_Inps_degrees : UDInt;
      END_STRUCT;
      read4 : Struct
         active_power : Array[1..3] of UDInt;
         active_power_tot : UDInt;
         reactive_power : Array[1..3] of UDInt;
         reactive_power_tot : UDInt;
         apparent_power : Array[1..3] of UDInt;
         apparent_power_tot : UDInt;
         power_factor : Array[1..3] of UDInt;
         power_factor_tot : UDInt;
      END_STRUCT;
      read6 : Struct
         fault_records : UDInt;
         event_records : UDInt;
         waveform_Records : UDInt;
         secondary_voltage : Array[1..3] of UDInt;
      END_STRUCT;
   END_VAR
BEGIN
   // Siemens - 7SR11 & 7SR12 - Argus - Overcurrent Relay
   // Energy Management
   //  
   // - https://cache.industry.siemens.com/dl/files/284/109747284/
   //   att_928907/v1/7SR12_Argus_Complete_Technical_Manual.pdf
   //   ==> page 212  

   "mb_station_block_header"(sb := #sb,
                             mb_query := #mb_query);
   #mb_query.mb_addr := #mb_addr;

   #mb_query.mode := #mb_query.c.mode.read;

   #mb_query(data_addr := 40010,
             data_ptr := #read1);
   IF #mb_query.Done THEN
       FOR #c := 1 TO 3 DO
           #out1.primary_Voltage_L_L[#c] := UDINT_TO_REAL(#read1.primary_Voltage_L_L[#c]) / 1000;
           #out1.primary_Voltage_L_N[#c] := UDINT_TO_REAL(#read1.primary_Voltage_L_N[#c]) / 1000;
           #out1.secondary_Voltage_L_N[#c] := UDINT_TO_REAL(#read1.secondary_Voltage_L_N[#c]) / 1000;
       END_FOR;
   END_IF;

   #mb_query(data_addr := 40034,
             data_ptr := #read2);
   IF #mb_query.Done THEN
       FOR #c := 1 TO 3 DO
           #out2.nominal_voltage_degrees_L_L[#c] := UDINT_TO_REAL(#read2.nominal_voltage_degrees_L_L[#c]) / 1000;
           #out2.nominal_voltage_degrees_L_N[#c] := UDINT_TO_REAL(#read2.nominal_voltage_degrees_L_N[#c]) / 1000;
       END_FOR;
       #out2.Vzps := UDINT_TO_REAL(#read2.Vzps) / 1000;
       #out2.Vpps := UDINT_TO_REAL(#read2.Vpps) / 1000;
       #out2.Vnps := UDINT_TO_REAL(#read2.Vnps) / 1000;
       #out2.Vzps_degree := UDINT_TO_REAL(#read2.Vzps_degree) / 1000;
       #out2.Vpps_degree := UDINT_TO_REAL(#read2.Vpps_degree) / 1000;
       #out2.Vnps_degree := UDINT_TO_REAL(#read2.Vnps_degree) / 1000;
       #out2.frequency := UDINT_TO_REAL(#read2.frequency) / 1000;
   END_IF;

   #mb_query(data_addr := 40064,
             data_ptr := #read3);
   IF #mb_query.Done THEN
       FOR #c := 1 TO 3 DO
           #out3.primary_current[#c] := UDINT_TO_REAL(#read3.primary_current[#c]) / 1000;
           #out3.secondary_current[#c] := UDINT_TO_REAL(#read3.secondary_current[#c]) / 1000;
           #out3.nominal_current[#c] := UDINT_TO_REAL(#read3.nominal_current[#c]) / 1000;
           #out3.nominal_current_degrees[#c] := UDINT_TO_REAL(#read3.nominal_current_degrees[#c]) / 1000;
       END_FOR;
       #out3.primary_In := UDINT_TO_REAL(#read3.primary_In) / 1000;
       #out3.secondary_In := UDINT_TO_REAL(#read3.secondary_In) / 1000;
       #out3.nominal_In := UDINT_TO_REAL(#read3.nominal_In) / 1000;
       #out3.primary_Ig := UDINT_TO_REAL(#read3.primary_Ig) / 1000;
       #out3.secondary_Ig := UDINT_TO_REAL(#read3.secondary_Ig) / 1000;
       #out3.nominal_Ig := UDINT_TO_REAL(#read3.nominal_Ig) / 1000;
       #out3.nominal_Izps := UDINT_TO_REAL(#read3.nominal_Izps) / 1000;
       #out3.nominal_Ipps := UDINT_TO_REAL(#read3.nominal_Ipps) / 1000;
       #out3.nominal_Inps := UDINT_TO_REAL(#read3.nominal_Inps) / 1000;
       #out3.nominal_Izps_degrees := UDINT_TO_REAL(#read3.nominal_Izps_degrees) / 1000;
       #out3.nominal_Ipps_degrees := UDINT_TO_REAL(#read3.nominal_Ipps_degrees) / 1000;
       #out3.nominal_Inps_degrees := UDINT_TO_REAL(#read3.nominal_Inps_degrees) / 1000;
   END_IF;

   #mb_query(data_addr := 40112,
             data_ptr := #read4);
   IF #mb_query.Done THEN
       FOR #c := 1 TO 3 DO
           #out4.active_power[#c] := UDINT_TO_REAL(#read4.active_power[#c]) / 1000;
           #out4.reactive_power[#c] := UDINT_TO_REAL(#read4.reactive_power[#c]) / 1000;
           #out4.apparent_power[#c] := UDINT_TO_REAL(#read4.apparent_power[#c]) / 1000;
           #out4.power_factor[#c] := UDINT_TO_REAL(#read4.power_factor[#c]) / 1000;
       END_FOR;
       #out4.active_power_tot := UDINT_TO_REAL(#read4.active_power_tot) / 1000;
       #out4.reactive_power_tot := UDINT_TO_REAL(#read4.reactive_power_tot) / 1000;
       #out4.apparent_power_tot := UDINT_TO_REAL(#read4.apparent_power_tot) / 1000;
       #out4.power_factor_tot := UDINT_TO_REAL(#read4.power_factor_tot) / 1000;
   END_IF;

   #mb_query(data_addr := 40144,
             data_ptr := #out5);

   #mb_query(data_addr := 40167,
             data_ptr := #read6);
   IF #mb_query.Done THEN
       FOR #c := 1 TO 3 DO
           #out6.secondary_voltage[#c] := UDINT_TO_REAL(#read6.secondary_voltage[#c]) / 1000;
       END_FOR;
       #out6.fault_records := UDINT_TO_REAL(#read6.fault_records) / 1000;
       #out6.event_records := UDINT_TO_REAL(#read6.event_records) / 1000;
       #out6.waveform_records := UDINT_TO_REAL(#read6.waveform_Records) / 1000;
   END_IF;

   "mb_station_block_footer"(sb := #sb,
                             mb_query := #mb_query);
END_FUNCTION_BLOCK

FUNCTION_BLOCK "Siemens_MAG_6000"   // FB54, SCL
{ S7_Optimized_Access := 'TRUE' }
VERSION : 0.1
   VAR_INPUT
      mb_addr : UInt;
   END_VAR
   VAR_IN_OUT
      mb_query : "mb_query";
   END_VAR
   VAR
      sb : "mb_station_block_udt";
      flow : Struct
         velocity : Real;   // mm/s
         flow : Real;
      END_STRUCT;
      totalizer : Array[1..3] of UDInt;
   END_VAR
BEGIN
   // Siemens - SITRANS F M MAG 6000

   "mb_station_block_header"(sb := #sb, mb_query := #mb_query);
   #mb_query.mb_addr := #mb_addr;

   #mb_query.mode := #mb_query.c.read.holding_reg;
   #mb_query(data_addr := 2999, data_ptr := #flow);
   #mb_query(data_addr := 3016, data_ptr := #totalizer);

   "mb_station_block_footer"(sb := #sb, mb_query := #mb_query);
END_FUNCTION_BLOCK

FUNCTION_BLOCK "Siemens_MASS_6000"   // FB55, SCL
{ S7_Optimized_Access := 'TRUE' }
VERSION : 0.1
   VAR_INPUT
      mb_addr : UInt;
   END_VAR
   VAR_IN_OUT
      mb_query : "mb_query";
   END_VAR
   VAR
      sb : "mb_station_block_udt";
      flow : Struct
         massflow : Real;   // [kg/s]
         volumeflow : Real;   // [m3/s]
         density : Real;   // [kg/m3]
         temperature : Real;   // [Â°C]
         fraction : Array[1..2] of Real;   // [kg/s]
         "%_fraction" : Real;   // [%]
         totalizer_1 : Array[1..2] of UDInt;   // [kg or m3]
         totalizer_2 : Array[1..2] of UDInt;   // [kg or m3]
         totalizer_real : Array[1..2] of Real;   // [kg or m3]
      END_STRUCT;
   END_VAR
BEGIN
   // Siemens - MASS 6000
   // https://cache.industry.siemens.com/dl/files/906/44880906/
   // att_70364/v1/USMII_MODBUS_AOM_OI_En_en-US.pdf

   "mb_station_block_header"(sb := #sb, mb_query := #mb_query);
   #mb_query.mb_addr := #mb_addr;

   #mb_query.mode := #mb_query.c.read.holding_reg;
   #mb_query(data_addr := 3000, data_ptr := #flow);

   "mb_station_block_footer"(sb := #sb, mb_query := #mb_query);
END_FUNCTION_BLOCK

FUNCTION_BLOCK "Siemens_sed2_modbus2"   // FB57, SCL
{ S7_Optimized_Access := 'TRUE' }
VERSION : 0.1
   VAR_INPUT
      mb_addr : UInt;
      ref : Real;   // 0-100% ( -100% reverse)
   END_VAR
   VAR_OUTPUT
      speed : Real;   // rpm
      current : Real;   // A x10
      torque : Real;   // Nm x10
      actual_pwr : Real;   // kW x100
      total_kwh : Real;   // kWh
      dc_bus_volt : Real;   // V
   END_VAR
   VAR_IN_OUT
      mb_query : "mb_query";
   END_VAR
   VAR
      sb : "mb_station_block_udt";
      write1 : Struct
         wdog_time : UInt := 1500;   // [ms]
         wdog_action : Word := 1;   // 1:stop, 0:no action
         freq_ref : UInt;
         run_enable : UInt;
         reverse : UInt;
         cmd_start : UInt;
         fault_ack : UInt;
      END_STRUCT;
      write2 : Struct
         current_limit : UInt := 4000;   // A x0
         accel_time : UInt := 1000;   // s x100
         decel_time : UInt := 1000;   // s x100
         manual : UInt;
      END_STRUCT;
      write3 : Struct
         freq_max : UInt := 5000;   // HZ x100
      END_STRUCT;
      read1 : Struct
         freq_output : UInt;   // Hz x10
         speed : UInt;   // rpm
         current : UInt;   // A x10
         torque : UInt;   // Nm x10
         actual_pwr : UInt;   // kW x100
         total_kwh : UInt;   // kWh
         dc_bus_volt : UInt;   // V
         reference : UInt;   // Hz x10
         rated_pwr : UInt;   // kWx100
         output_volts : UInt;
         reverse : UInt;
         run : UInt;
         at_max_freq : UInt;
         ctrl_mode : UInt;   // 1:SERIAL, 0:LOCAL
         enabled : UInt;
         ready_to_run : UInt;
         analog_in_1 : UInt;
         analog_in_2 : UInt;
      END_STRUCT;
      read2 : Struct
         digital_in : Array[1..6] of UInt;
         fault : UInt;
         last_fault : UInt;
         fault_hist : Array[1..4] of UInt;
         warning : UInt;
         last_warning : UInt;
      END_STRUCT;
   END_VAR
   VAR_TEMP
      "real" : Real;
   END_VAR
BEGIN
   // Siemens - SED2-MODBUS2 - Variable Frequency Drive
   // Modbus RTU Interface Module for SED2 
   // 
   // https://www.downloads.siemens.com/download-center/
   // Download.aspx?pos=download&fct=getasset&id1=A6V10073869

   #write1.reverse := BOOL_TO_UINT(#ref < 0);
   #"real" := NORM_X(MIN := 0, VALUE := #ref, MAX := ABS(100));
   #write1.freq_ref := SCALE_X(MIN := 0, VALUE := #"real", MAX := 16#4000);
   #write1.run_enable := BOOL_TO_UINT(#ref <> 0);
   #write1.cmd_start := BOOL_TO_UINT(#ref <> 0);

   "mb_station_block_header"(sb := #sb,
                             mb_query := #mb_query);
   #mb_query.mb_addr := #mb_addr;

   #mb_query.mode := #mb_query.c.mode.write;
   #mb_query(data_addr := 40001,
             data_ptr := #write1);
   #mb_query(data_addr := 40010,
             data_ptr := #write2);
   #mb_query(data_addr := 40016,
             data_ptr := #write3);

   #mb_query.mode := #mb_query.c.mode.read;
   #mb_query(data_addr := 40024,
             data_ptr := #read1);
   #mb_query(data_addr := 40048,
             data_ptr := #read2);

   "mb_station_block_footer"(sb := #sb,
                             mb_query := #mb_query);

   #speed := UINT_TO_REAL(#read1.speed);
   #current := UINT_TO_REAL(#read1.current) / 10;
   #torque := UINT_TO_REAL(#read1.torque) / 10;
   #actual_pwr := UINT_TO_REAL(#read1.actual_pwr) / 100;
   #total_kwh := UINT_TO_REAL(#read1.total_kwh);
   #dc_bus_volt := UINT_TO_REAL(#read1.dc_bus_volt);
END_FUNCTION_BLOCK

FUNCTION_BLOCK "Siemens_Sinamics_G120"   // FB58, SCL
{ S7_Optimized_Access := 'TRUE' }
VERSION : 0.1
   VAR_INPUT
      mb_addr : UInt;
      ref : Real;
   END_VAR
   VAR_IN_OUT
      mb_query : "mb_query";
   END_VAR
   VAR
      sb : "mb_station_block_udt";
      read : Struct
         stw : Struct
            x08_Speed_setpoint : Bool;   // Actual value deviation within tolerance t_off
            x09_Control_requested : Bool;
            x10_f_or_n_comparison_value_reached_exceeded : Bool;
            x11_I_M_or_P_limit_not_reached : Bool;
            x12 : Bool;
            x13_No_motor_overtemperature_alarm : Bool;
            x14_Motor_rotates_forwards : Bool;   // 0 = Motor rotates backwards (n_act < 0)
            x15_No_alarm_thermal_overload_power_unit : Bool;
            x00_Ready_to_power_up : Bool;
            x01_Ready_to_operate : Bool;   // (DC link loaded, pulses blocked)
            x02_Operation_enabled : Bool;   // (drive follows n_set)
            x03_Fault_present : Bool;
            x04_No_coast_down_active : Bool;   // (OFF2 inactive)
            x05_No_fast_stop_active : Bool;   // (OFF3 inactive)
            x06_power_on_inhibit_active : Bool;
            x07_Alarm_present : Bool;
         END_STRUCT;
         actual : Int;
      END_STRUCT;
      write : Struct
         ctw : Struct
            x08 : Bool;
            x09 : Bool;
            x10_control_via_PLC : Bool := TRUE;
            x11_reversal : Bool;
            x12 : Bool;
            x13_Motorized_potentiometer_setpoint_raise : Bool;
            x14_Motorized_potentiometer_setpoint_lower : Bool;
            x15 : Bool;
            x00_R_TRIG_ON : Bool;   // 0 = OFF1 (braking with ramp-function generator, then pulse cancllation &ready-to-power-up)
            x01_No_OFF2 : Bool := TRUE;   // enable is possible. 0 = OFF2 (immediate pulse cancellation and power-on inhibit)
            x02_No_OFF3 : Bool := TRUE;   // enable is possible. 0 = OFF3 braking with the OFF3 ramp p1135, then pulse cancellation andpower-on inhibit)
            x03_Enable_operation : Bool := TRUE;   // (pulses can be enabled) 0 = Inhibit operation (cancel pulses)
            x04_Operating_condition : Bool;   // (the ramp-function generator can be enabled)0 = Inhibit ramp-function generator (set the ramp-function generator output tozero)
            x05_Enable_the_ramp_function_generator : Bool;   // 0 = Stop the ramp-function generator (freeze the ramp-function generatoroutput)
            x06_enable_setpoint : Bool := TRUE;   // 0 = Inhibit setpoint (set the ramp-function generator input to zero)
            x07_R_TRIG_acknowledge_faults : Bool;
         END_STRUCT;
         setpoint : Int;
      END_STRUCT;
   END_VAR
BEGIN
   // Siemens - SINAMICS G120
   // 
   // Web: https://cache.industry.siemens.com/dl/files/944/
   // 35928944/att_7966/v1/application_cu230_modbus_v1_2_en.pdf

   "mb_station_block_header"(sb := #sb, mb_query := #mb_query);
   #mb_query.mb_addr := #mb_addr;

   #mb_query.mode := #mb_query.c.read.holding_reg;
   #mb_query(data_addr := 40110, data_ptr := #read);

   #write.ctw.x00_R_TRIG_ON :=
   (* *)#ref <> 0
   (* *)AND NOT #read.stw.x07_Alarm_present
   (* *)AND #read.stw.x01_Ready_to_operate
   (* *)AND #read.stw.x00_Ready_to_power_up;
   #write.setpoint := REAL_TO_INT(#ref);

   #mb_query.mode := #mb_query.c.write.holding_reg;
   #mb_query(data_addr := 40100, data_ptr := #write);

   "mb_station_block_footer"(sb := #sb, mb_query := #mb_query);
END_FUNCTION_BLOCK

FUNCTION_BLOCK "Siemens_SITRANS_F_M_MAG_8000"   // FB59, SCL
{ S7_Optimized_Access := 'TRUE' }
VERSION : 0.1
   VAR_INPUT
      mb_addr : UInt;
   END_VAR
   VAR_IN_OUT
      mb_query : "mb_query";
   END_VAR
   VAR
      sb : "mb_station_block_udt";
      flow : Struct
         velocity : Real;   // mm/s
         flow : Real;
      END_STRUCT;
      totalizer : Array[1..3] of UDInt;
   END_VAR
BEGIN
   // Siemens - SITRANS F M MAG 8000
   // https://cache.industry.siemens.com/dl/files/509/54091509/
   // att_100244/v1/A5E03409989_01_MAG8000_MODBUS_AOM_OI_.pdf

   "mb_station_block_header"(sb := #sb, mb_query := #mb_query);
   #mb_query.mb_addr := #mb_addr;

   #mb_query.mode := #mb_query.c.read.holding_reg;
   #mb_query(data_addr := 2999, data_ptr := #flow);
   #mb_query(data_addr := 3016, data_ptr := #totalizer);

   "mb_station_block_footer"(sb := #sb, mb_query := #mb_query);
END_FUNCTION_BLOCK

